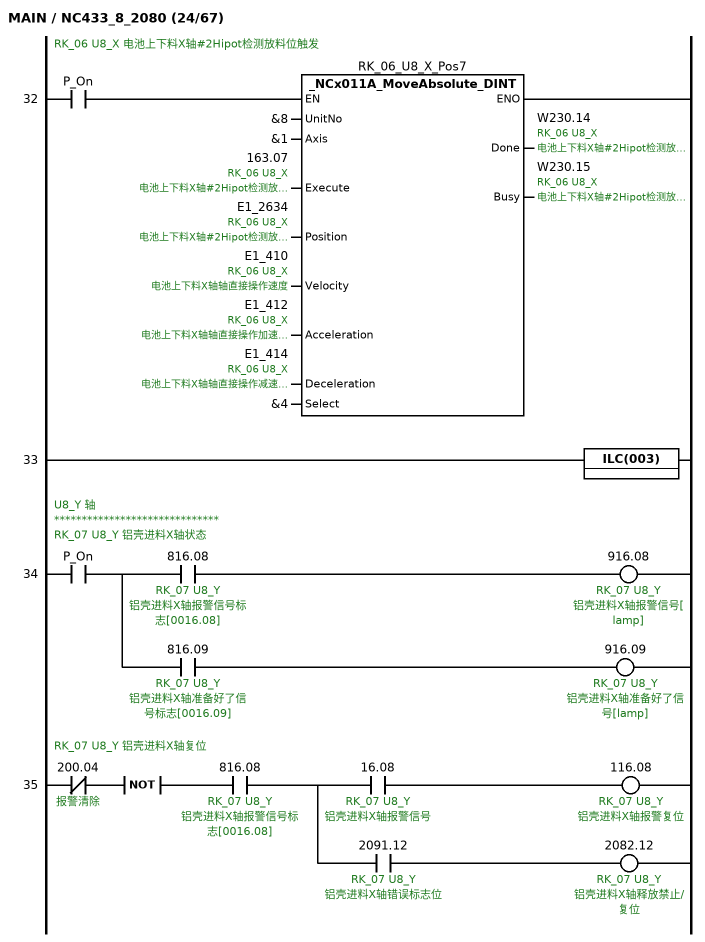
; [picture p288: MAIN / NC433_8_2080, rungs 32-35]
; rung 32: RK_06 U8_X 电池上下料X轴#2Hipot检测放料位触发
LD P_On
CALL RK_06_U8_X_Pos7 : _NCx011A_MoveAbsolute_DINT (UnitNo := &8, Axis := &1, Execute := 163.07, Position := E1_2634, Velocity := E1_410, Acceleration := E1_412, Deceleration := E1_414, Select := &4, Done => W230.14, Busy => W230.15)  ; RK_06 U8_X 电池上下料X轴#2Hipot检测放料位触发, RK_06 U8_X 电池上下料X轴#2Hipot检测放料位, RK_06 U8_X 电池上下料X轴轴直接操作速度, RK_06 U8_X 电池上下料X轴轴直接操作加速时间, RK_06 U8_X 电池上下料X轴轴直接操作减速时间, RK_06 U8_X 电池上下料X轴#2Hipot检测放料位完成标志, RK_06 U8_X 电池上下料X轴#2Hipot检测放料位忙标志
; rung 33
ILC(003)
; rung 34: U8_Y 轴 / ****************************** / RK_07 U8_Y 铝壳进料X轴状态
LD P_On
OUT TR0
AND 816.08  ; RK_07 U8_Y 铝壳进料X轴报警信号标志[0016.08]
OUT 916.08  ; RK_07 U8_Y 铝壳进料X轴报警信号[lamp]
LD TR0
AND 816.09  ; RK_07 U8_Y 铝壳进料X轴准备好了信号标志[0016.09]
OUT 916.09  ; RK_07 U8_Y 铝壳进料X轴准备好了信号[lamp]
; rung 35: RK_07 U8_Y 铝壳进料X轴复位
LDNOT 200.04  ; 报警清除
NOT(520)
AND 816.08  ; RK_07 U8_Y 铝壳进料X轴报警信号标志[0016.08]
OUT TR0
AND 16.08  ; RK_07 U8_Y 铝壳进料X轴报警信号
OUT 116.08  ; RK_07 U8_Y 铝壳进料X轴报警复位
LD TR0
AND 2091.12  ; RK_07 U8_Y 铝壳进料X轴错误标志位
OUT 2082.12  ; RK_07 U8_Y 铝壳进料X轴释放禁止/复位

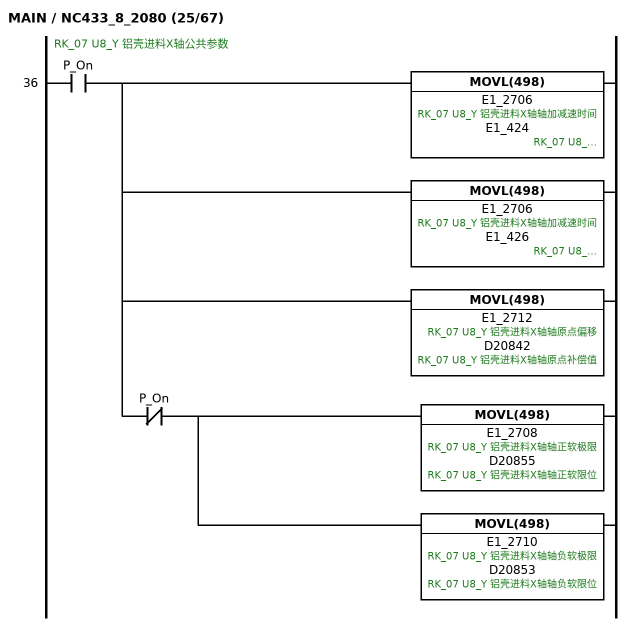
; rung 36: RK_07 U8_Y 铝壳进料X轴公共参数
LD P_On
MOVL(498) E1_2706 E1_424  ; RK_07 U8_Y 铝壳进料X轴轴加减速时间, RK_07 U8_Y 铝壳进料X轴轴直接操作加速时间
MOVL(498) E1_2706 E1_426  ; RK_07 U8_Y 铝壳进料X轴轴加减速时间, RK_07 U8_Y 铝壳进料X轴轴直接操作减速时间
MOVL(498) E1_2712 D20842  ; RK_07 U8_Y 铝壳进料X轴轴原点偏移, RK_07 U8_Y 铝壳进料X轴轴原点补偿值
ANDNOT P_On
MOVL(498) E1_2708 D20855  ; RK_07 U8_Y 铝壳进料X轴轴正软极限, RK_07 U8_Y 铝壳进料X轴轴正软限位
MOVL(498) E1_2710 D20853  ; RK_07 U8_Y 铝壳进料X轴轴负软极限, RK_07 U8_Y 铝壳进料X轴轴负软限位

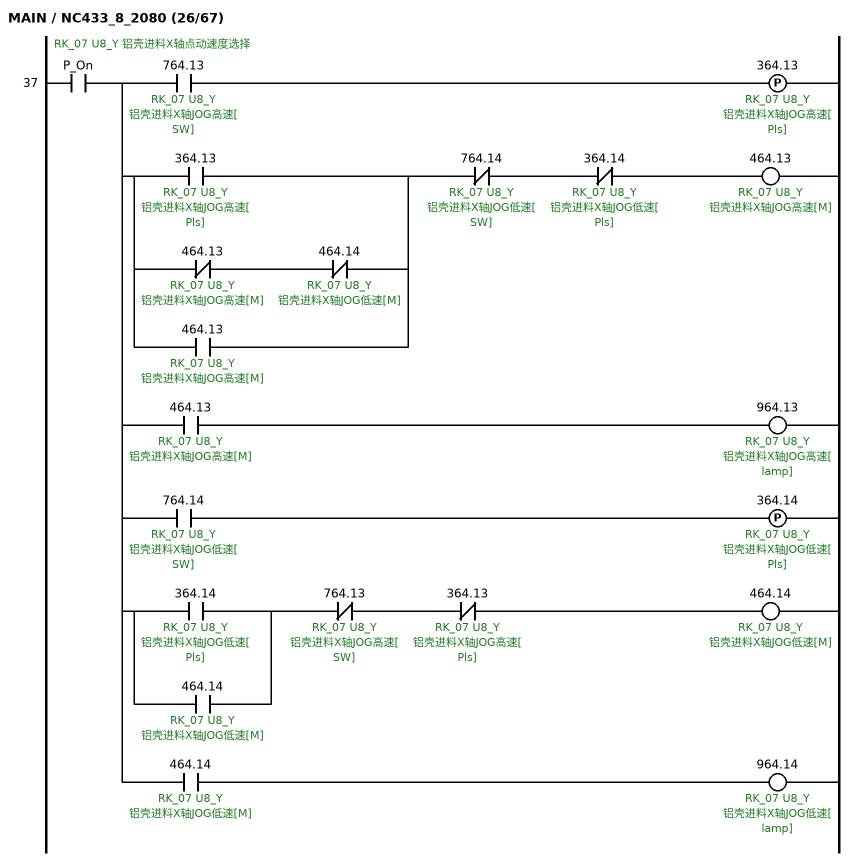
; rung 37: RK_07 U8_Y 铝壳进料X轴点动速度选择
LD P_On
OUT TR0
AND 764.13  ; RK_07 U8_Y 铝壳进料X轴JOG高速[SW]
DIFU(013) 364.13  ; RK_07 U8_Y 铝壳进料X轴JOG高速[Pls]
LD TR0
LD 364.13  ; RK_07 U8_Y 铝壳进料X轴JOG高速[Pls]
LDNOT 464.13  ; RK_07 U8_Y 铝壳进料X轴JOG高速[M]
ANDNOT 464.14  ; RK_07 U8_Y 铝壳进料X轴JOG低速[M]
ORLD
OR 464.13  ; RK_07 U8_Y 铝壳进料X轴JOG高速[M]
ANDLD
ANDNOT 764.14  ; RK_07 U8_Y 铝壳进料X轴JOG低速[SW]
ANDNOT 364.14  ; RK_07 U8_Y 铝壳进料X轴JOG低速[Pls]
OUT 464.13  ; RK_07 U8_Y 铝壳进料X轴JOG高速[M]
LD TR0
AND 464.13  ; RK_07 U8_Y 铝壳进料X轴JOG高速[M]
OUT 964.13  ; RK_07 U8_Y 铝壳进料X轴JOG高速[lamp]
LD TR0
AND 764.14  ; RK_07 U8_Y 铝壳进料X轴JOG低速[SW]
DIFU(013) 364.14  ; RK_07 U8_Y 铝壳进料X轴JOG低速[Pls]
LD TR0
LD 364.14  ; RK_07 U8_Y 铝壳进料X轴JOG低速[Pls]
OR 464.14  ; RK_07 U8_Y 铝壳进料X轴JOG低速[M]
ANDLD
ANDNOT 764.13  ; RK_07 U8_Y 铝壳进料X轴JOG高速[SW]
ANDNOT 364.13  ; RK_07 U8_Y 铝壳进料X轴JOG高速[Pls]
OUT 464.14  ; RK_07 U8_Y 铝壳进料X轴JOG低速[M]
LD TR0
AND 464.14  ; RK_07 U8_Y 铝壳进料X轴JOG低速[M]
OUT 964.14  ; RK_07 U8_Y 铝壳进料X轴JOG低速[lamp]

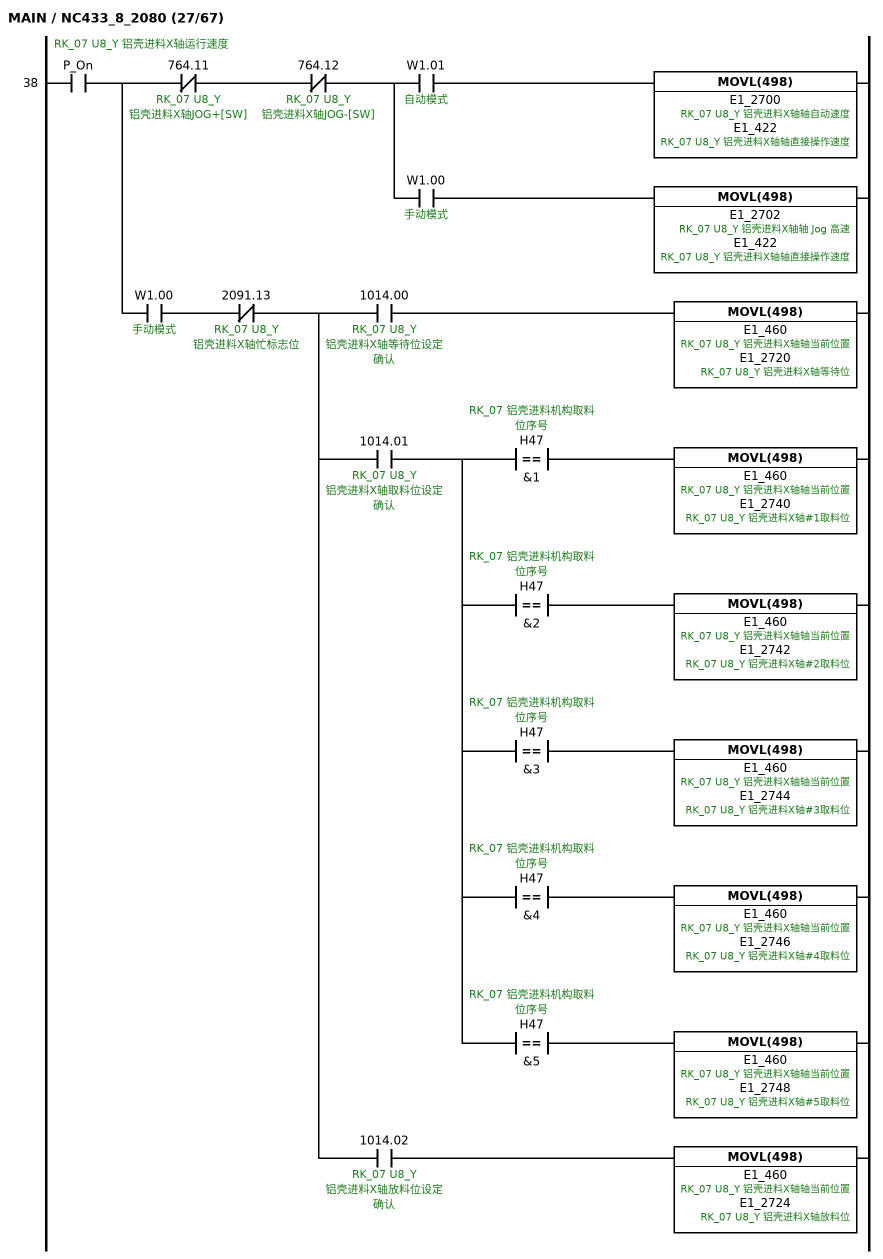
; rung 38: RK_07 U8_Y 铝壳进料X轴运行速度
LD P_On
OUT TR0
ANDNOT 764.11  ; RK_07 U8_Y 铝壳进料X轴JOG+[SW]
ANDNOT 764.12  ; RK_07 U8_Y 铝壳进料X轴JOG-[SW]
OUT TR1
AND W1.01  ; 自动模式
MOVL(498) E1_2700 E1_422  ; RK_07 U8_Y 铝壳进料X轴轴自动速度, RK_07 U8_Y 铝壳进料X轴轴直接操作速度
LD TR1
AND W1.00  ; 手动模式
MOVL(498) E1_2702 E1_422  ; RK_07 U8_Y 铝壳进料X轴轴 Jog 高速, RK_07 U8_Y 铝壳进料X轴轴直接操作速度
LD TR0
AND W1.00  ; 手动模式
ANDNOT 2091.13  ; RK_07 U8_Y 铝壳进料X轴忙标志位
OUT TR0
AND 1014.00  ; RK_07 U8_Y 铝壳进料X轴等待位设定确认
MOVL(498) E1_460 E1_2720  ; RK_07 U8_Y 铝壳进料X轴轴当前位置, RK_07 U8_Y 铝壳进料X轴等待位
LD TR0
AND 1014.01  ; RK_07 U8_Y 铝壳进料X轴取料位设定确认
OUT TR1
AND=(300) H47 &1  ; RK_07 铝壳进料机构取料位序号
MOVL(498) E1_460 E1_2740  ; RK_07 U8_Y 铝壳进料X轴轴当前位置, RK_07 U8_Y 铝壳进料X轴#1取料位
LD TR1
AND=(300) H47 &2  ; RK_07 铝壳进料机构取料位序号
MOVL(498) E1_460 E1_2742  ; RK_07 U8_Y 铝壳进料X轴轴当前位置, RK_07 U8_Y 铝壳进料X轴#2取料位
LD TR1
AND=(300) H47 &3  ; RK_07 铝壳进料机构取料位序号
MOVL(498) E1_460 E1_2744  ; RK_07 U8_Y 铝壳进料X轴轴当前位置, RK_07 U8_Y 铝壳进料X轴#3取料位
LD TR1
AND=(300) H47 &4  ; RK_07 铝壳进料机构取料位序号
MOVL(498) E1_460 E1_2746  ; RK_07 U8_Y 铝壳进料X轴轴当前位置, RK_07 U8_Y 铝壳进料X轴#4取料位
LD TR1
AND=(300) H47 &5  ; RK_07 铝壳进料机构取料位序号
MOVL(498) E1_460 E1_2748  ; RK_07 U8_Y 铝壳进料X轴轴当前位置, RK_07 U8_Y 铝壳进料X轴#5取料位
LD TR0
AND 1014.02  ; RK_07 U8_Y 铝壳进料X轴放料位设定确认
MOVL(498) E1_460 E1_2724  ; RK_07 U8_Y 铝壳进料X轴轴当前位置, RK_07 U8_Y 铝壳进料X轴放料位

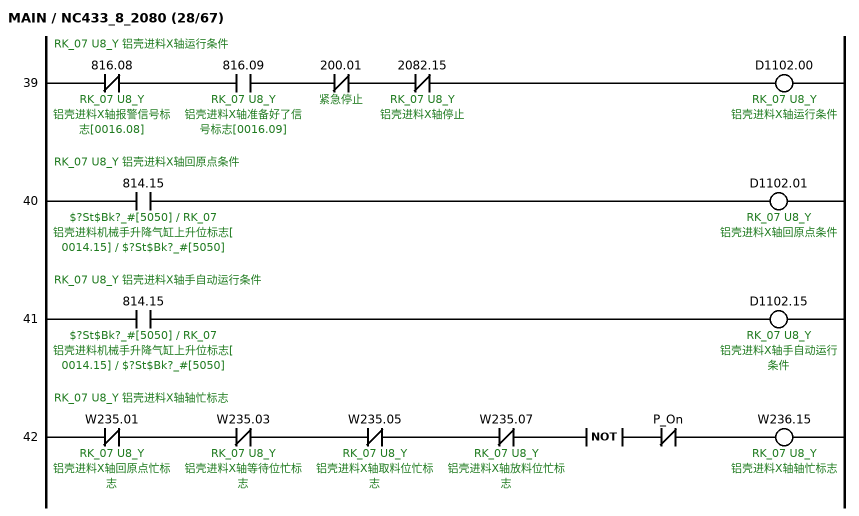
; rung 39: RK_07 U8_Y 铝壳进料X轴运行条件
LDNOT 816.08  ; RK_07 U8_Y 铝壳进料X轴报警信号标志[0016.08]
AND 816.09  ; RK_07 U8_Y 铝壳进料X轴准备好了信号标志[0016.09]
ANDNOT 200.01  ; 紧急停止
ANDNOT 2082.15  ; RK_07 U8_Y 铝壳进料X轴停止
OUT D1102.00  ; RK_07 U8_Y 铝壳进料X轴运行条件
; rung 40: RK_07 U8_Y 铝壳进料X轴回原点条件
LD 814.15  ; $?St$Bk?_#[5050] / RK_07 铝壳进料机械手升降气缸上升位标志[0014.15] / $?St$Bk?_#[5050]
OUT D1102.01  ; RK_07 U8_Y 铝壳进料X轴回原点条件
; rung 41: RK_07 U8_Y 铝壳进料X轴手自动运行条件
LD 814.15  ; $?St$Bk?_#[5050] / RK_07 铝壳进料机械手升降气缸上升位标志[0014.15] / $?St$Bk?_#[5050]
OUT D1102.15  ; RK_07 U8_Y 铝壳进料X轴手自动运行条件
; rung 42: RK_07 U8_Y 铝壳进料X轴轴忙标志
LDNOT W235.01  ; RK_07 U8_Y 铝壳进料X轴回原点忙标志
ANDNOT W235.03  ; RK_07 U8_Y 铝壳进料X轴等待位忙标志
ANDNOT W235.05  ; RK_07 U8_Y 铝壳进料X轴取料位忙标志
ANDNOT W235.07  ; RK_07 U8_Y 铝壳进料X轴放料位忙标志
NOT(520)
ANDNOT P_On
OUT W236.15  ; RK_07 U8_Y 铝壳进料X轴轴忙标志

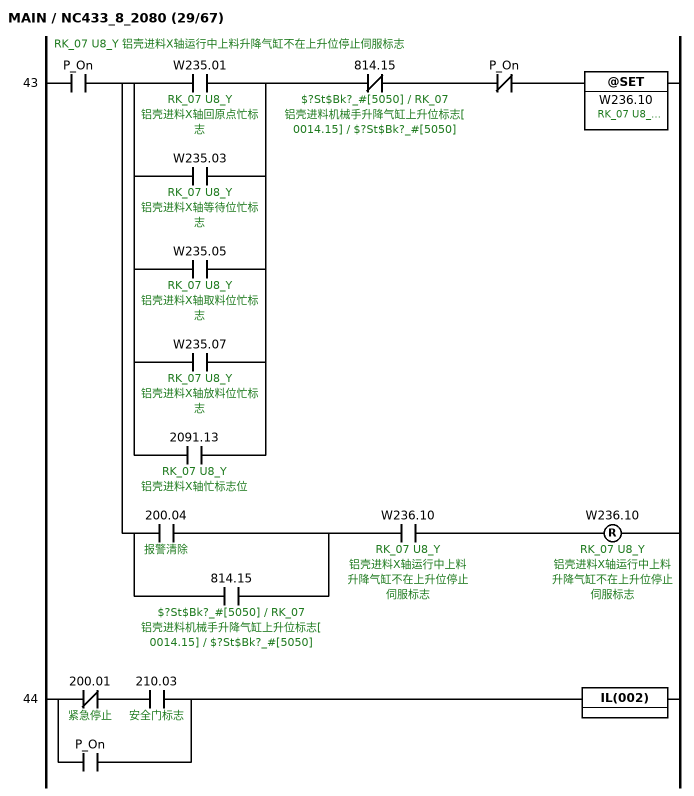
; rung 43: RK_07 U8_Y 铝壳进料X轴运行中上料升降气缸不在上升位停止伺服标志
LD P_On
OUT TR0
LD W235.01  ; RK_07 U8_Y 铝壳进料X轴回原点忙标志
OR W235.03  ; RK_07 U8_Y 铝壳进料X轴等待位忙标志
OR W235.05  ; RK_07 U8_Y 铝壳进料X轴取料位忙标志
OR W235.07  ; RK_07 U8_Y 铝壳进料X轴放料位忙标志
OR 2091.13  ; RK_07 U8_Y 铝壳进料X轴忙标志位
ANDLD
ANDNOT 814.15  ; $?St$Bk?_#[5050] / RK_07 铝壳进料机械手升降气缸上升位标志[0014.15] / $?St$Bk?_#[5050]
ANDNOT P_On
@SET W236.10  ; RK_07 U8_Y 铝壳进料X轴运行中上料升降气缸不在上升位停止伺服标志  // 增加相应报警信息
LD TR0
LD 200.04  ; 报警清除
OR 814.15  ; $?St$Bk?_#[5050] / RK_07 铝壳进料机械手升降气缸上升位标志[0014.15] / $?St$Bk?_#[5050]
ANDLD
AND W236.10  ; RK_07 U8_Y 铝壳进料X轴运行中上料升降气缸不在上升位停止伺服标志
RSET W236.10  ; RK_07 U8_Y 铝壳进料X轴运行中上料升降气缸不在上升位停止伺服标志
; rung 44
LDNOT 200.01  ; 紧急停止
AND 210.03  ; 安全门标志
OR P_On
IL(002)

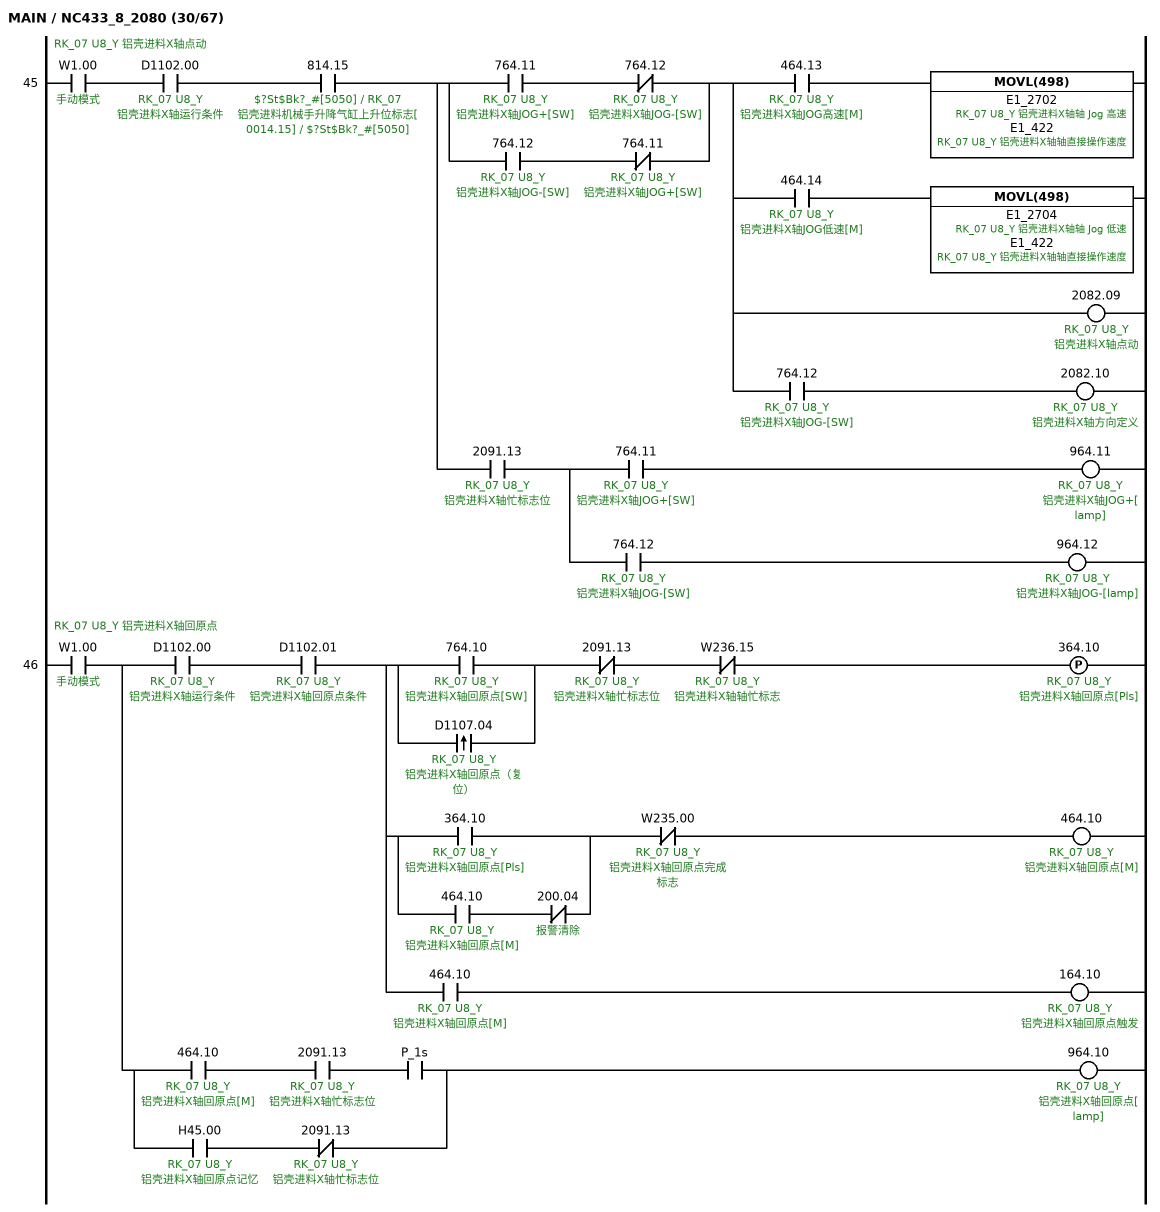
; rung 45: RK_07 U8_Y 铝壳进料X轴点动
LD W1.00  ; 手动模式
AND D1102.00  ; RK_07 U8_Y 铝壳进料X轴运行条件
AND 814.15  ; $?St$Bk?_#[5050] / RK_07 铝壳进料机械手升降气缸上升位标志[0014.15] / $?St$Bk?_#[5050]
OUT TR0
LD 764.11  ; RK_07 U8_Y 铝壳进料X轴JOG+[SW]
ANDNOT 764.12  ; RK_07 U8_Y 铝壳进料X轴JOG-[SW]
LD 764.12  ; RK_07 U8_Y 铝壳进料X轴JOG-[SW]
ANDNOT 764.11  ; RK_07 U8_Y 铝壳进料X轴JOG+[SW]
ORLD
ANDLD
OUT TR1
AND 464.13  ; RK_07 U8_Y 铝壳进料X轴JOG高速[M]
MOVL(498) E1_2702 E1_422  ; RK_07 U8_Y 铝壳进料X轴轴 Jog 高速, RK_07 U8_Y 铝壳进料X轴轴直接操作速度
LD TR1
AND 464.14  ; RK_07 U8_Y 铝壳进料X轴JOG低速[M]
MOVL(498) E1_2704 E1_422  ; RK_07 U8_Y 铝壳进料X轴轴 Jog 低速, RK_07 U8_Y 铝壳进料X轴轴直接操作速度
LD TR1
OUT 2082.09  ; RK_07 U8_Y 铝壳进料X轴点动
AND 764.12  ; RK_07 U8_Y 铝壳进料X轴JOG-[SW]
OUT 2082.10  ; RK_07 U8_Y 铝壳进料X轴方向定义
LD TR0
AND 2091.13  ; RK_07 U8_Y 铝壳进料X轴忙标志位
OUT TR0
AND 764.11  ; RK_07 U8_Y 铝壳进料X轴JOG+[SW]
OUT 964.11  ; RK_07 U8_Y 铝壳进料X轴JOG+[lamp]
LD TR0
AND 764.12  ; RK_07 U8_Y 铝壳进料X轴JOG-[SW]
OUT 964.12  ; RK_07 U8_Y 铝壳进料X轴JOG-[lamp]
; rung 46: RK_07 U8_Y 铝壳进料X轴回原点
LD W1.00  ; 手动模式
OUT TR0
AND D1102.00  ; RK_07 U8_Y 铝壳进料X轴运行条件
AND D1102.01  ; RK_07 U8_Y 铝壳进料X轴回原点条件
OUT TR1
LD 764.10  ; RK_07 U8_Y 铝壳进料X轴回原点[SW]
@OR D1107.04  ; RK_07 U8_Y 铝壳进料X轴回原点（复位）
ANDLD
ANDNOT 2091.13  ; RK_07 U8_Y 铝壳进料X轴忙标志位
ANDNOT W236.15  ; RK_07 U8_Y 铝壳进料X轴轴忙标志
DIFU(013) 364.10  ; RK_07 U8_Y 铝壳进料X轴回原点[Pls]
LD TR1
LD 364.10  ; RK_07 U8_Y 铝壳进料X轴回原点[Pls]
LD 464.10  ; RK_07 U8_Y 铝壳进料X轴回原点[M]
ANDNOT 200.04  ; 报警清除
ORLD
ANDLD
ANDNOT W235.00  ; RK_07 U8_Y 铝壳进料X轴回原点完成标志
OUT 464.10  ; RK_07 U8_Y 铝壳进料X轴回原点[M]
LD TR1
AND 464.10  ; RK_07 U8_Y 铝壳进料X轴回原点[M]
OUT 164.10  ; RK_07 U8_Y 铝壳进料X轴回原点触发
LD TR0
LD 464.10  ; RK_07 U8_Y 铝壳进料X轴回原点[M]
AND 2091.13  ; RK_07 U8_Y 铝壳进料X轴忙标志位
AND P_1s
LD H45.00  ; RK_07 U8_Y 铝壳进料X轴回原点记忆
ANDNOT 2091.13  ; RK_07 U8_Y 铝壳进料X轴忙标志位
ORLD
ANDLD
OUT 964.10  ; RK_07 U8_Y 铝壳进料X轴回原点[lamp]

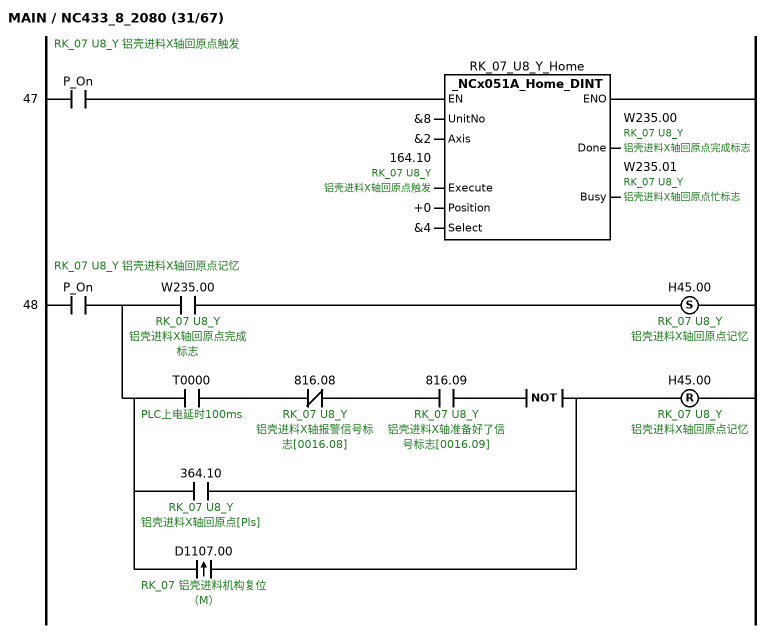
; rung 47: RK_07 U8_Y 铝壳进料X轴回原点触发
LD P_On
CALL RK_07_U8_Y_Home : _NCx051A_Home_DINT (UnitNo := &8, Axis := &2, Execute := 164.10, Position := +0, Select := &4, Done => W235.00, Busy => W235.01)  ; RK_07 U8_Y 铝壳进料X轴回原点触发, RK_07 U8_Y 铝壳进料X轴回原点完成标志, RK_07 U8_Y 铝壳进料X轴回原点忙标志
; rung 48: RK_07 U8_Y 铝壳进料X轴回原点记忆
LD P_On
OUT TR0
AND W235.00  ; RK_07 U8_Y 铝壳进料X轴回原点完成标志
SET H45.00  ; RK_07 U8_Y 铝壳进料X轴回原点记忆
LD TR0
LD T0000  ; PLC上电延时100ms
ANDNOT 816.08  ; RK_07 U8_Y 铝壳进料X轴报警信号标志[0016.08]
AND 816.09  ; RK_07 U8_Y 铝壳进料X轴准备好了信号标志[0016.09]
NOT(520)
OR 364.10  ; RK_07 U8_Y 铝壳进料X轴回原点[Pls]
@OR D1107.00  ; RK_07 铝壳进料机构复位（M）
ANDLD
RSET H45.00  ; RK_07 U8_Y 铝壳进料X轴回原点记忆

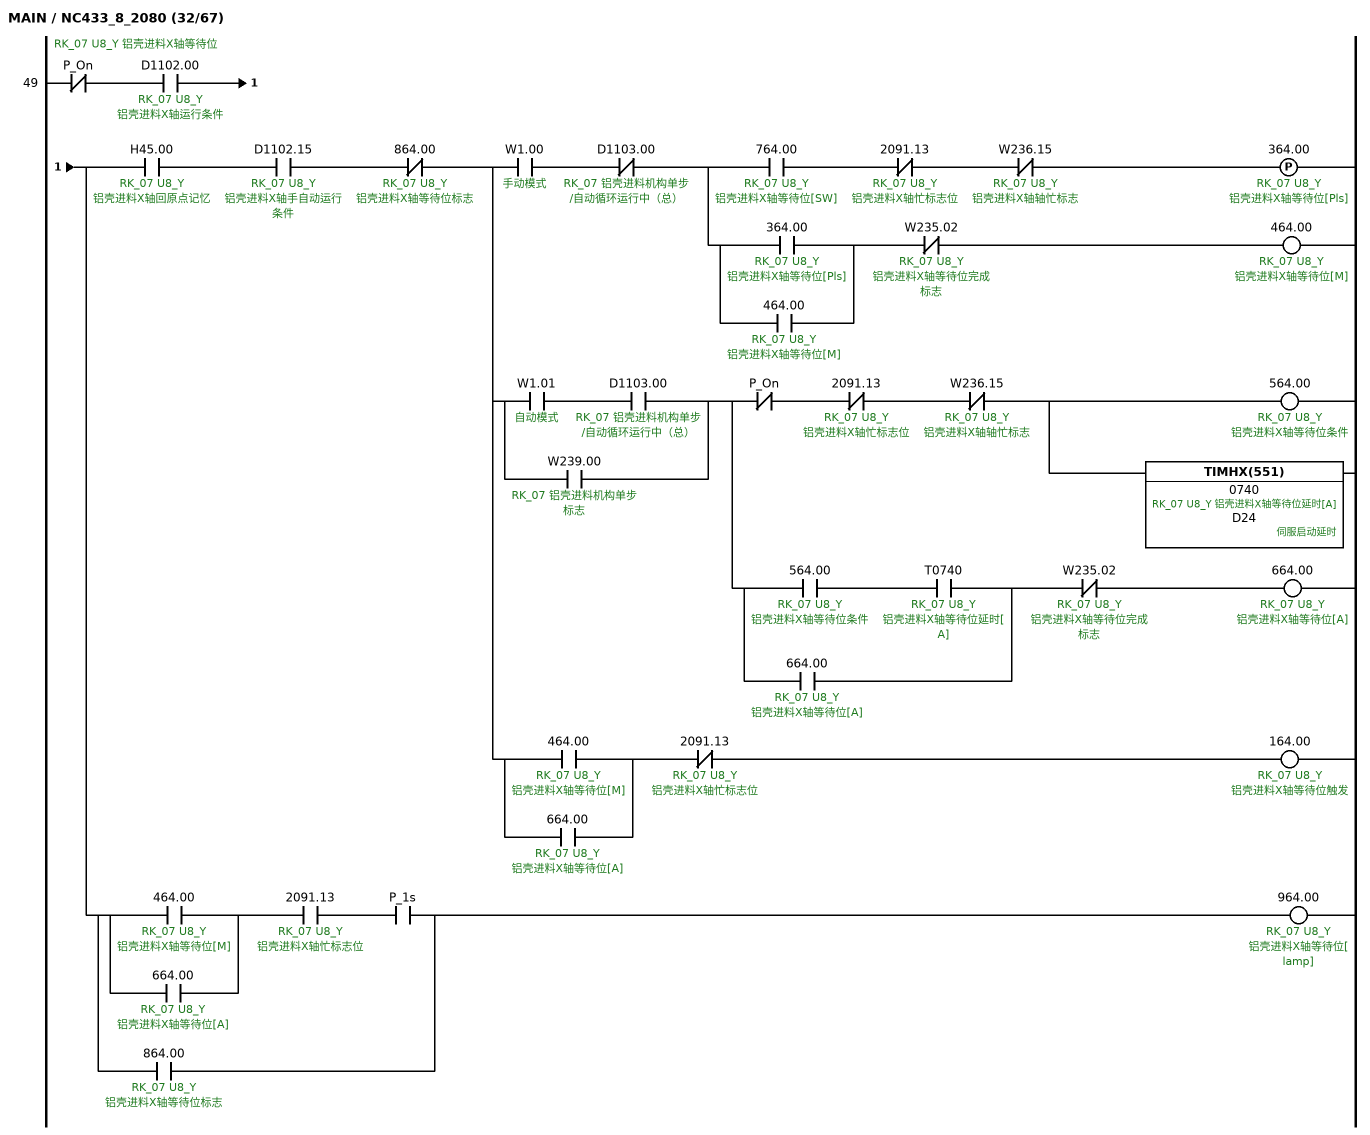
; rung 49: RK_07 U8_Y 铝壳进料X轴等待位
LDNOT P_On
AND D1102.00  ; RK_07 U8_Y 铝壳进料X轴运行条件
OUT TR0
AND H45.00  ; RK_07 U8_Y 铝壳进料X轴回原点记忆
AND D1102.15  ; RK_07 U8_Y 铝壳进料X轴手自动运行条件
ANDNOT 864.00  ; RK_07 U8_Y 铝壳进料X轴等待位标志
OUT TR1
AND W1.00  ; 手动模式
ANDNOT D1103.00  ; RK_07 铝壳进料机构单步/自动循环运行中（总）
OUT TR2
AND 764.00  ; RK_07 U8_Y 铝壳进料X轴等待位[SW]
ANDNOT 2091.13  ; RK_07 U8_Y 铝壳进料X轴忙标志位
ANDNOT W236.15  ; RK_07 U8_Y 铝壳进料X轴轴忙标志
DIFU(013) 364.00  ; RK_07 U8_Y 铝壳进料X轴等待位[Pls]
LD TR2
LD 364.00  ; RK_07 U8_Y 铝壳进料X轴等待位[Pls]
OR 464.00  ; RK_07 U8_Y 铝壳进料X轴等待位[M]
ANDLD
ANDNOT W235.02  ; RK_07 U8_Y 铝壳进料X轴等待位完成标志
OUT 464.00  ; RK_07 U8_Y 铝壳进料X轴等待位[M]
LD TR1
LD W1.01  ; 自动模式
AND D1103.00  ; RK_07 铝壳进料机构单步/自动循环运行中（总）
OR W239.00  ; RK_07 铝壳进料机构单步标志
ANDLD
OUT TR2
ANDNOT P_On  // RK_07 U8_Y 铝壳进料X轴等待位（步）
ANDNOT 2091.13  ; RK_07 U8_Y 铝壳进料X轴忙标志位
ANDNOT W236.15  ; RK_07 U8_Y 铝壳进料X轴轴忙标志
OUT 564.00  ; RK_07 U8_Y 铝壳进料X轴等待位条件
TIMHX(551) 0740 D24  ; 伺服启动延时, RK_07 U8_Y 铝壳进料X轴等待位延时[A]
LD TR2
LD 564.00  ; RK_07 U8_Y 铝壳进料X轴等待位条件
AND T0740  ; RK_07 U8_Y 铝壳进料X轴等待位延时[A]
OR 664.00  ; RK_07 U8_Y 铝壳进料X轴等待位[A]
ANDLD
ANDNOT W235.02  ; RK_07 U8_Y 铝壳进料X轴等待位完成标志
OUT 664.00  ; RK_07 U8_Y 铝壳进料X轴等待位[A]
LD TR1
LD 464.00  ; RK_07 U8_Y 铝壳进料X轴等待位[M]
OR 664.00  ; RK_07 U8_Y 铝壳进料X轴等待位[A]
ANDLD
ANDNOT 2091.13  ; RK_07 U8_Y 铝壳进料X轴忙标志位
OUT 164.00  ; RK_07 U8_Y 铝壳进料X轴等待位触发
LD TR0
LD 464.00  ; RK_07 U8_Y 铝壳进料X轴等待位[M]
OR 664.00  ; RK_07 U8_Y 铝壳进料X轴等待位[A]
AND 2091.13  ; RK_07 U8_Y 铝壳进料X轴忙标志位
AND P_1s
OR 864.00  ; RK_07 U8_Y 铝壳进料X轴等待位标志
ANDLD
OUT 964.00  ; RK_07 U8_Y 铝壳进料X轴等待位[lamp]

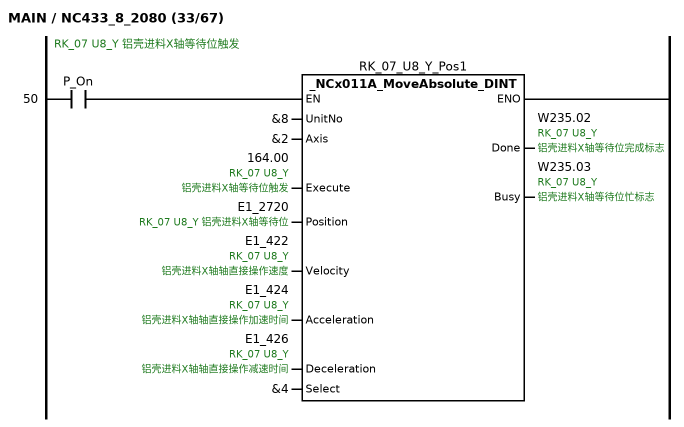
; rung 50: RK_07 U8_Y 铝壳进料X轴等待位触发
LD P_On
CALL RK_07_U8_Y_Pos1 : _NCx011A_MoveAbsolute_DINT (UnitNo := &8, Axis := &2, Execute := 164.00, Position := E1_2720, Velocity := E1_422, Acceleration := E1_424, Deceleration := E1_426, Select := &4, Done => W235.02, Busy => W235.03)  ; RK_07 U8_Y 铝壳进料X轴等待位触发, RK_07 U8_Y 铝壳进料X轴等待位, RK_07 U8_Y 铝壳进料X轴轴直接操作速度, RK_07 U8_Y 铝壳进料X轴轴直接操作加速时间, RK_07 U8_Y 铝壳进料X轴轴直接操作减速时间, RK_07 U8_Y 铝壳进料X轴等待位完成标志, RK_07 U8_Y 铝壳进料X轴等待位忙标志

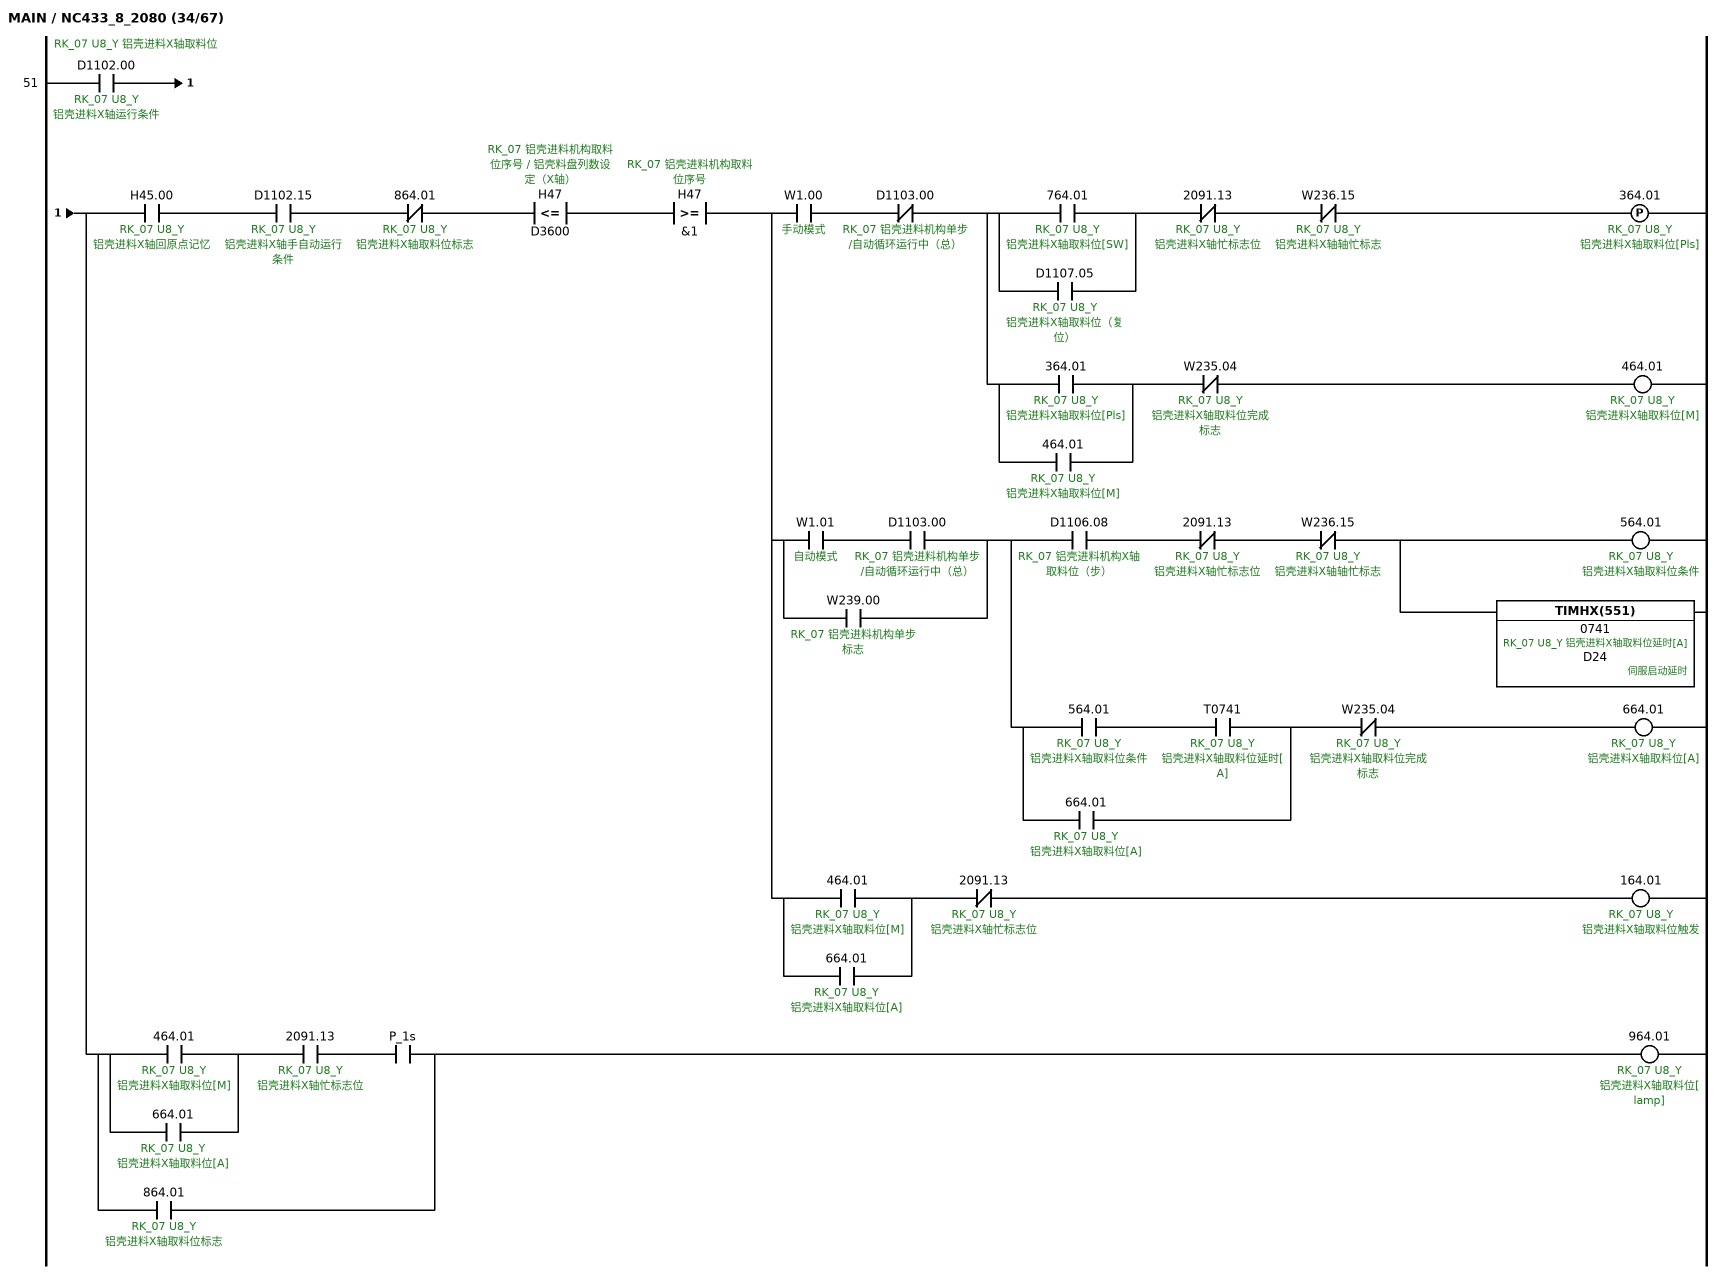
; rung 51: RK_07 U8_Y 铝壳进料X轴取料位
LD D1102.00  ; RK_07 U8_Y 铝壳进料X轴运行条件
OUT TR0
AND H45.00  ; RK_07 U8_Y 铝壳进料X轴回原点记忆
AND D1102.15  ; RK_07 U8_Y 铝壳进料X轴手自动运行条件
ANDNOT 864.01  ; RK_07 U8_Y 铝壳进料X轴取料位标志
AND<=(315) H47 D3600  ; RK_07 铝壳进料机构取料位序号, 铝壳料盘列数设定（X轴）
AND>=(325) H47 &1  ; RK_07 铝壳进料机构取料位序号
OUT TR1
AND W1.00  ; 手动模式
ANDNOT D1103.00  ; RK_07 铝壳进料机构单步/自动循环运行中（总）
OUT TR2
LD 764.01  ; RK_07 U8_Y 铝壳进料X轴取料位[SW]
OR D1107.05  ; RK_07 U8_Y 铝壳进料X轴取料位（复位）
ANDLD
ANDNOT 2091.13  ; RK_07 U8_Y 铝壳进料X轴忙标志位
ANDNOT W236.15  ; RK_07 U8_Y 铝壳进料X轴轴忙标志
DIFU(013) 364.01  ; RK_07 U8_Y 铝壳进料X轴取料位[Pls]
LD TR2
LD 364.01  ; RK_07 U8_Y 铝壳进料X轴取料位[Pls]
OR 464.01  ; RK_07 U8_Y 铝壳进料X轴取料位[M]
ANDLD
ANDNOT W235.04  ; RK_07 U8_Y 铝壳进料X轴取料位完成标志
OUT 464.01  ; RK_07 U8_Y 铝壳进料X轴取料位[M]
LD TR1
LD W1.01  ; 自动模式
AND D1103.00  ; RK_07 铝壳进料机构单步/自动循环运行中（总）
OR W239.00  ; RK_07 铝壳进料机构单步标志
ANDLD
OUT TR2
AND D1106.08  ; RK_07 铝壳进料机构X轴取料位（步）
ANDNOT 2091.13  ; RK_07 U8_Y 铝壳进料X轴忙标志位
ANDNOT W236.15  ; RK_07 U8_Y 铝壳进料X轴轴忙标志
OUT 564.01  ; RK_07 U8_Y 铝壳进料X轴取料位条件
TIMHX(551) 0741 D24  ; 伺服启动延时, RK_07 U8_Y 铝壳进料X轴取料位延时[A]
LD TR2
LD 564.01  ; RK_07 U8_Y 铝壳进料X轴取料位条件
AND T0741  ; RK_07 U8_Y 铝壳进料X轴取料位延时[A]
OR 664.01  ; RK_07 U8_Y 铝壳进料X轴取料位[A]
ANDLD
ANDNOT W235.04  ; RK_07 U8_Y 铝壳进料X轴取料位完成标志
OUT 664.01  ; RK_07 U8_Y 铝壳进料X轴取料位[A]
LD TR1
LD 464.01  ; RK_07 U8_Y 铝壳进料X轴取料位[M]
OR 664.01  ; RK_07 U8_Y 铝壳进料X轴取料位[A]
ANDLD
ANDNOT 2091.13  ; RK_07 U8_Y 铝壳进料X轴忙标志位
OUT 164.01  ; RK_07 U8_Y 铝壳进料X轴取料位触发
LD TR0
LD 464.01  ; RK_07 U8_Y 铝壳进料X轴取料位[M]
OR 664.01  ; RK_07 U8_Y 铝壳进料X轴取料位[A]
AND 2091.13  ; RK_07 U8_Y 铝壳进料X轴忙标志位
AND P_1s
OR 864.01  ; RK_07 U8_Y 铝壳进料X轴取料位标志
ANDLD
OUT 964.01  ; RK_07 U8_Y 铝壳进料X轴取料位[lamp]

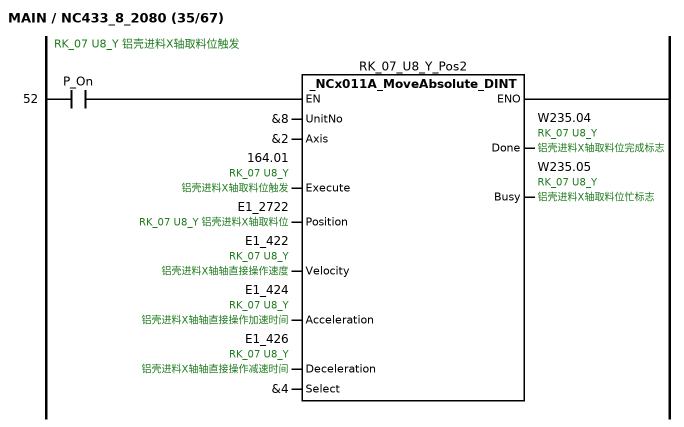
; rung 52: RK_07 U8_Y 铝壳进料X轴取料位触发
LD P_On
CALL RK_07_U8_Y_Pos2 : _NCx011A_MoveAbsolute_DINT (UnitNo := &8, Axis := &2, Execute := 164.01, Position := E1_2722, Velocity := E1_422, Acceleration := E1_424, Deceleration := E1_426, Select := &4, Done => W235.04, Busy => W235.05)  ; RK_07 U8_Y 铝壳进料X轴取料位触发, RK_07 U8_Y 铝壳进料X轴取料位, RK_07 U8_Y 铝壳进料X轴轴直接操作速度, RK_07 U8_Y 铝壳进料X轴轴直接操作加速时间, RK_07 U8_Y 铝壳进料X轴轴直接操作减速时间, RK_07 U8_Y 铝壳进料X轴取料位完成标志, RK_07 U8_Y 铝壳进料X轴取料位忙标志

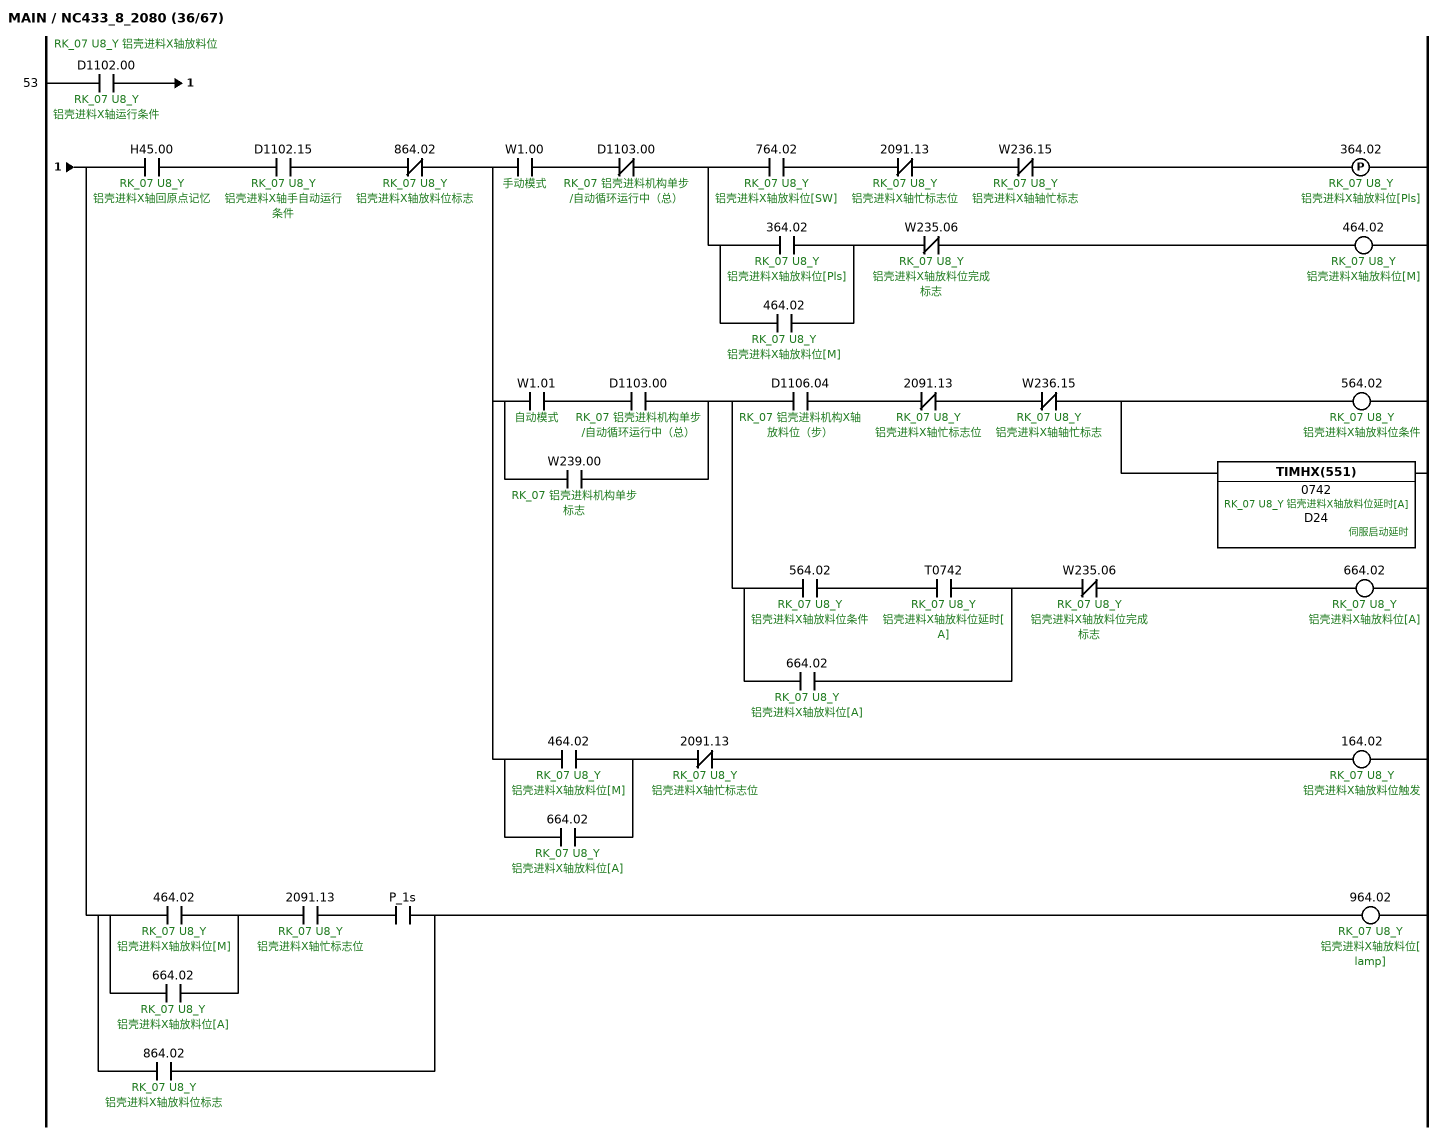
; rung 53: RK_07 U8_Y 铝壳进料X轴放料位
LD D1102.00  ; RK_07 U8_Y 铝壳进料X轴运行条件
OUT TR0
AND H45.00  ; RK_07 U8_Y 铝壳进料X轴回原点记忆
AND D1102.15  ; RK_07 U8_Y 铝壳进料X轴手自动运行条件
ANDNOT 864.02  ; RK_07 U8_Y 铝壳进料X轴放料位标志
OUT TR1
AND W1.00  ; 手动模式
ANDNOT D1103.00  ; RK_07 铝壳进料机构单步/自动循环运行中（总）
OUT TR2
AND 764.02  ; RK_07 U8_Y 铝壳进料X轴放料位[SW]
ANDNOT 2091.13  ; RK_07 U8_Y 铝壳进料X轴忙标志位
ANDNOT W236.15  ; RK_07 U8_Y 铝壳进料X轴轴忙标志
DIFU(013) 364.02  ; RK_07 U8_Y 铝壳进料X轴放料位[Pls]
LD TR2
LD 364.02  ; RK_07 U8_Y 铝壳进料X轴放料位[Pls]
OR 464.02  ; RK_07 U8_Y 铝壳进料X轴放料位[M]
ANDLD
ANDNOT W235.06  ; RK_07 U8_Y 铝壳进料X轴放料位完成标志
OUT 464.02  ; RK_07 U8_Y 铝壳进料X轴放料位[M]
LD TR1
LD W1.01  ; 自动模式
AND D1103.00  ; RK_07 铝壳进料机构单步/自动循环运行中（总）
OR W239.00  ; RK_07 铝壳进料机构单步标志
ANDLD
OUT TR2
AND D1106.04  ; RK_07 铝壳进料机构X轴放料位（步）
ANDNOT 2091.13  ; RK_07 U8_Y 铝壳进料X轴忙标志位
ANDNOT W236.15  ; RK_07 U8_Y 铝壳进料X轴轴忙标志
OUT 564.02  ; RK_07 U8_Y 铝壳进料X轴放料位条件
TIMHX(551) 0742 D24  ; 伺服启动延时, RK_07 U8_Y 铝壳进料X轴放料位延时[A]
LD TR2
LD 564.02  ; RK_07 U8_Y 铝壳进料X轴放料位条件
AND T0742  ; RK_07 U8_Y 铝壳进料X轴放料位延时[A]
OR 664.02  ; RK_07 U8_Y 铝壳进料X轴放料位[A]
ANDLD
ANDNOT W235.06  ; RK_07 U8_Y 铝壳进料X轴放料位完成标志
OUT 664.02  ; RK_07 U8_Y 铝壳进料X轴放料位[A]
LD TR1
LD 464.02  ; RK_07 U8_Y 铝壳进料X轴放料位[M]
OR 664.02  ; RK_07 U8_Y 铝壳进料X轴放料位[A]
ANDLD
ANDNOT 2091.13  ; RK_07 U8_Y 铝壳进料X轴忙标志位
OUT 164.02  ; RK_07 U8_Y 铝壳进料X轴放料位触发
LD TR0
LD 464.02  ; RK_07 U8_Y 铝壳进料X轴放料位[M]
OR 664.02  ; RK_07 U8_Y 铝壳进料X轴放料位[A]
AND 2091.13  ; RK_07 U8_Y 铝壳进料X轴忙标志位
AND P_1s
OR 864.02  ; RK_07 U8_Y 铝壳进料X轴放料位标志
ANDLD
OUT 964.02  ; RK_07 U8_Y 铝壳进料X轴放料位[lamp]

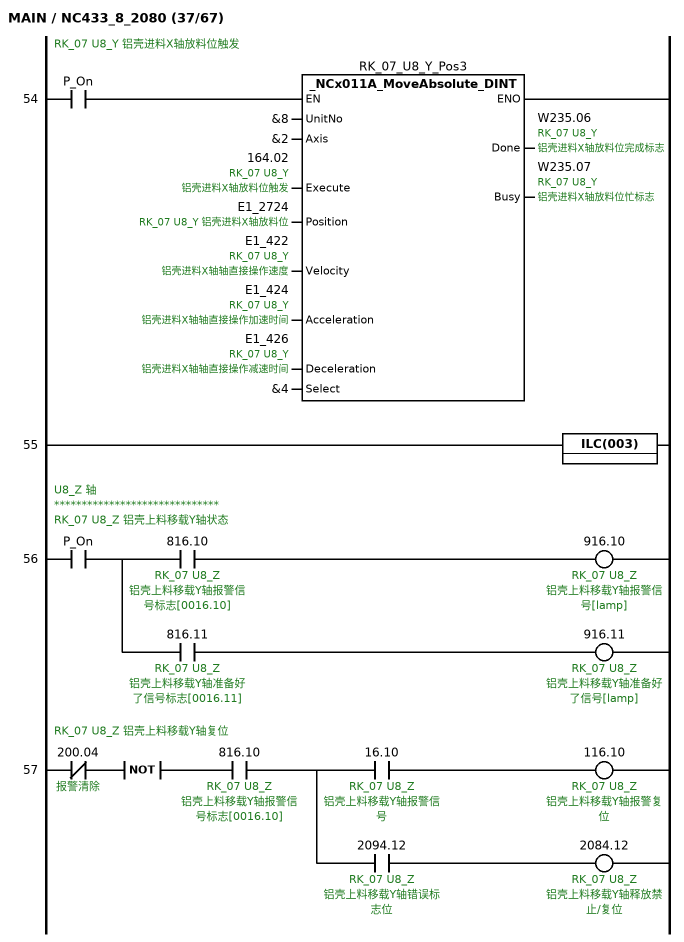
; rung 54: RK_07 U8_Y 铝壳进料X轴放料位触发
LD P_On
CALL RK_07_U8_Y_Pos3 : _NCx011A_MoveAbsolute_DINT (UnitNo := &8, Axis := &2, Execute := 164.02, Position := E1_2724, Velocity := E1_422, Acceleration := E1_424, Deceleration := E1_426, Select := &4, Done => W235.06, Busy => W235.07)  ; RK_07 U8_Y 铝壳进料X轴放料位触发, RK_07 U8_Y 铝壳进料X轴放料位, RK_07 U8_Y 铝壳进料X轴轴直接操作速度, RK_07 U8_Y 铝壳进料X轴轴直接操作加速时间, RK_07 U8_Y 铝壳进料X轴轴直接操作减速时间, RK_07 U8_Y 铝壳进料X轴放料位完成标志, RK_07 U8_Y 铝壳进料X轴放料位忙标志
; rung 55
ILC(003)
; rung 56: U8_Z 轴 / ****************************** / RK_07 U8_Z 铝壳上料移载Y轴状态
LD P_On
OUT TR0
AND 816.10  ; RK_07 U8_Z 铝壳上料移载Y轴报警信号标志[0016.10]
OUT 916.10  ; RK_07 U8_Z 铝壳上料移载Y轴报警信号[lamp]
LD TR0
AND 816.11  ; RK_07 U8_Z 铝壳上料移载Y轴准备好了信号标志[0016.11]
OUT 916.11  ; RK_07 U8_Z 铝壳上料移载Y轴准备好了信号[lamp]
; rung 57: RK_07 U8_Z 铝壳上料移载Y轴复位
LDNOT 200.04  ; 报警清除
NOT(520)
AND 816.10  ; RK_07 U8_Z 铝壳上料移载Y轴报警信号标志[0016.10]
OUT TR0
AND 16.10  ; RK_07 U8_Z 铝壳上料移载Y轴报警信号
OUT 116.10  ; RK_07 U8_Z 铝壳上料移载Y轴报警复位
LD TR0
AND 2094.12  ; RK_07 U8_Z 铝壳上料移载Y轴错误标志位
OUT 2084.12  ; RK_07 U8_Z 铝壳上料移载Y轴释放禁止/复位

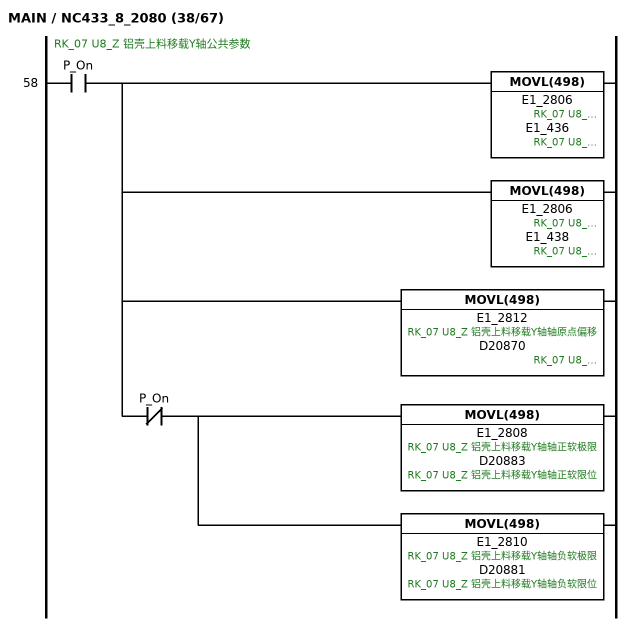
; rung 58: RK_07 U8_Z 铝壳上料移载Y轴公共参数
LD P_On
MOVL(498) E1_2806 E1_436  ; RK_07 U8_Z 铝壳上料移载Y轴轴加减速时间, RK_07 U8_Z 铝壳上料移载Y轴轴直接操作加速时间
MOVL(498) E1_2806 E1_438  ; RK_07 U8_Z 铝壳上料移载Y轴轴加减速时间, RK_07 U8_Z 铝壳上料移载Y轴轴直接操作减速时间
MOVL(498) E1_2812 D20870  ; RK_07 U8_Z 铝壳上料移载Y轴轴原点偏移, RK_07 U8_Z 铝壳上料移载Y轴轴原点补偿值
ANDNOT P_On
MOVL(498) E1_2808 D20883  ; RK_07 U8_Z 铝壳上料移载Y轴轴正软极限, RK_07 U8_Z 铝壳上料移载Y轴轴正软限位
MOVL(498) E1_2810 D20881  ; RK_07 U8_Z 铝壳上料移载Y轴轴负软极限, RK_07 U8_Z 铝壳上料移载Y轴轴负软限位

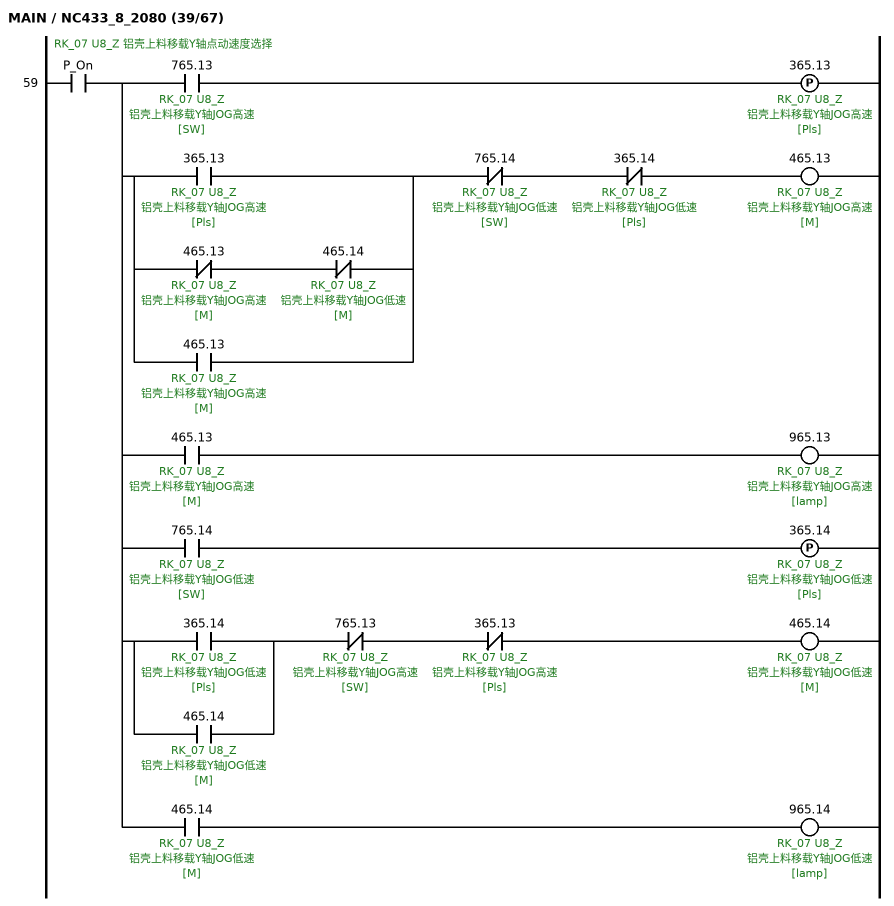
; rung 59: RK_07 U8_Z 铝壳上料移载Y轴点动速度选择
LD P_On
OUT TR0
AND 765.13  ; RK_07 U8_Z 铝壳上料移载Y轴JOG高速[SW]
DIFU(013) 365.13  ; RK_07 U8_Z 铝壳上料移载Y轴JOG高速[Pls]
LD TR0
LD 365.13  ; RK_07 U8_Z 铝壳上料移载Y轴JOG高速[Pls]
LDNOT 465.13  ; RK_07 U8_Z 铝壳上料移载Y轴JOG高速[M]
ANDNOT 465.14  ; RK_07 U8_Z 铝壳上料移载Y轴JOG低速[M]
ORLD
OR 465.13  ; RK_07 U8_Z 铝壳上料移载Y轴JOG高速[M]
ANDLD
ANDNOT 765.14  ; RK_07 U8_Z 铝壳上料移载Y轴JOG低速[SW]
ANDNOT 365.14  ; RK_07 U8_Z 铝壳上料移载Y轴JOG低速[Pls]
OUT 465.13  ; RK_07 U8_Z 铝壳上料移载Y轴JOG高速[M]
LD TR0
AND 465.13  ; RK_07 U8_Z 铝壳上料移载Y轴JOG高速[M]
OUT 965.13  ; RK_07 U8_Z 铝壳上料移载Y轴JOG高速[lamp]
LD TR0
AND 765.14  ; RK_07 U8_Z 铝壳上料移载Y轴JOG低速[SW]
DIFU(013) 365.14  ; RK_07 U8_Z 铝壳上料移载Y轴JOG低速[Pls]
LD TR0
LD 365.14  ; RK_07 U8_Z 铝壳上料移载Y轴JOG低速[Pls]
OR 465.14  ; RK_07 U8_Z 铝壳上料移载Y轴JOG低速[M]
ANDLD
ANDNOT 765.13  ; RK_07 U8_Z 铝壳上料移载Y轴JOG高速[SW]
ANDNOT 365.13  ; RK_07 U8_Z 铝壳上料移载Y轴JOG高速[Pls]
OUT 465.14  ; RK_07 U8_Z 铝壳上料移载Y轴JOG低速[M]
LD TR0
AND 465.14  ; RK_07 U8_Z 铝壳上料移载Y轴JOG低速[M]
OUT 965.14  ; RK_07 U8_Z 铝壳上料移载Y轴JOG低速[lamp]

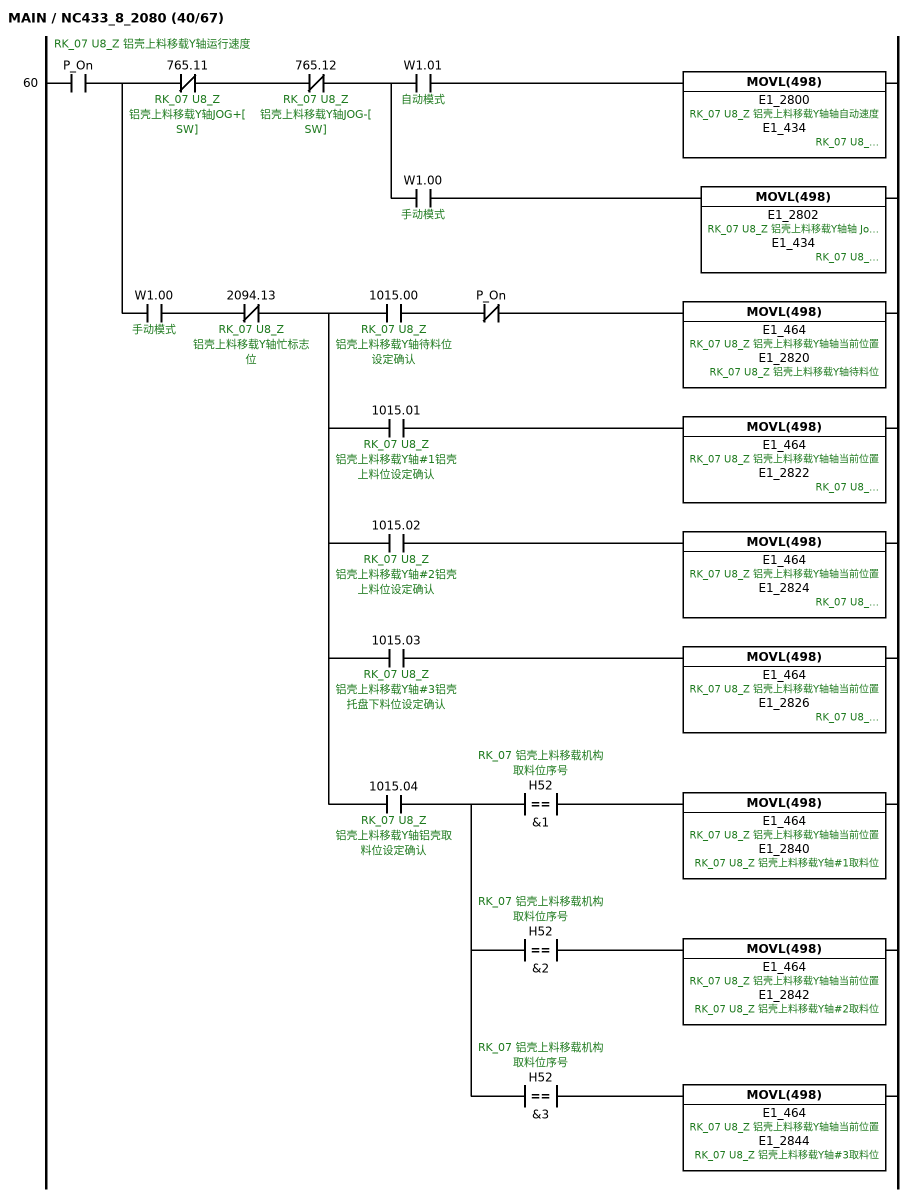
; rung 60: RK_07 U8_Z 铝壳上料移载Y轴运行速度
LD P_On
OUT TR0
ANDNOT 765.11  ; RK_07 U8_Z 铝壳上料移载Y轴JOG+[SW]
ANDNOT 765.12  ; RK_07 U8_Z 铝壳上料移载Y轴JOG-[SW]
OUT TR1
AND W1.01  ; 自动模式
MOVL(498) E1_2800 E1_434  ; RK_07 U8_Z 铝壳上料移载Y轴轴自动速度, RK_07 U8_Z 铝壳上料移载Y轴轴直接操作速度
LD TR1
AND W1.00  ; 手动模式
MOVL(498) E1_2802 E1_434  ; RK_07 U8_Z 铝壳上料移载Y轴轴 Jog 高速, RK_07 U8_Z 铝壳上料移载Y轴轴直接操作速度
LD TR0
AND W1.00  ; 手动模式
ANDNOT 2094.13  ; RK_07 U8_Z 铝壳上料移载Y轴忙标志位
OUT TR0
AND 1015.00  ; RK_07 U8_Z 铝壳上料移载Y轴待料位设定确认
ANDNOT P_On
MOVL(498) E1_464 E1_2820  ; RK_07 U8_Z 铝壳上料移载Y轴轴当前位置, RK_07 U8_Z 铝壳上料移载Y轴待料位
LD TR0
AND 1015.01  ; RK_07 U8_Z 铝壳上料移载Y轴#1铝壳上料位设定确认
MOVL(498) E1_464 E1_2822  ; RK_07 U8_Z 铝壳上料移载Y轴轴当前位置, RK_07 U8_Z 铝壳上料移载Y轴#1铝壳上料位
LD TR0
AND 1015.02  ; RK_07 U8_Z 铝壳上料移载Y轴#2铝壳上料位设定确认
MOVL(498) E1_464 E1_2824  ; RK_07 U8_Z 铝壳上料移载Y轴轴当前位置, RK_07 U8_Z 铝壳上料移载Y轴#2铝壳上料位
LD TR0
AND 1015.03  ; RK_07 U8_Z 铝壳上料移载Y轴#3铝壳托盘下料位设定确认
MOVL(498) E1_464 E1_2826  ; RK_07 U8_Z 铝壳上料移载Y轴轴当前位置, RK_07 U8_Z 铝壳上料移载Y轴#3铝壳托盘下料位
LD TR0
AND 1015.04  ; RK_07 U8_Z 铝壳上料移载Y轴铝壳取料位设定确认
OUT TR0
AND=(300) H52 &1  ; RK_07 铝壳上料移载机构取料位序号
MOVL(498) E1_464 E1_2840  ; RK_07 U8_Z 铝壳上料移载Y轴轴当前位置, RK_07 U8_Z 铝壳上料移载Y轴#1取料位
LD TR0
AND=(300) H52 &2  ; RK_07 铝壳上料移载机构取料位序号
MOVL(498) E1_464 E1_2842  ; RK_07 U8_Z 铝壳上料移载Y轴轴当前位置, RK_07 U8_Z 铝壳上料移载Y轴#2取料位
LD TR0
AND=(300) H52 &3  ; RK_07 铝壳上料移载机构取料位序号
MOVL(498) E1_464 E1_2844  ; RK_07 U8_Z 铝壳上料移载Y轴轴当前位置, RK_07 U8_Z 铝壳上料移载Y轴#3取料位

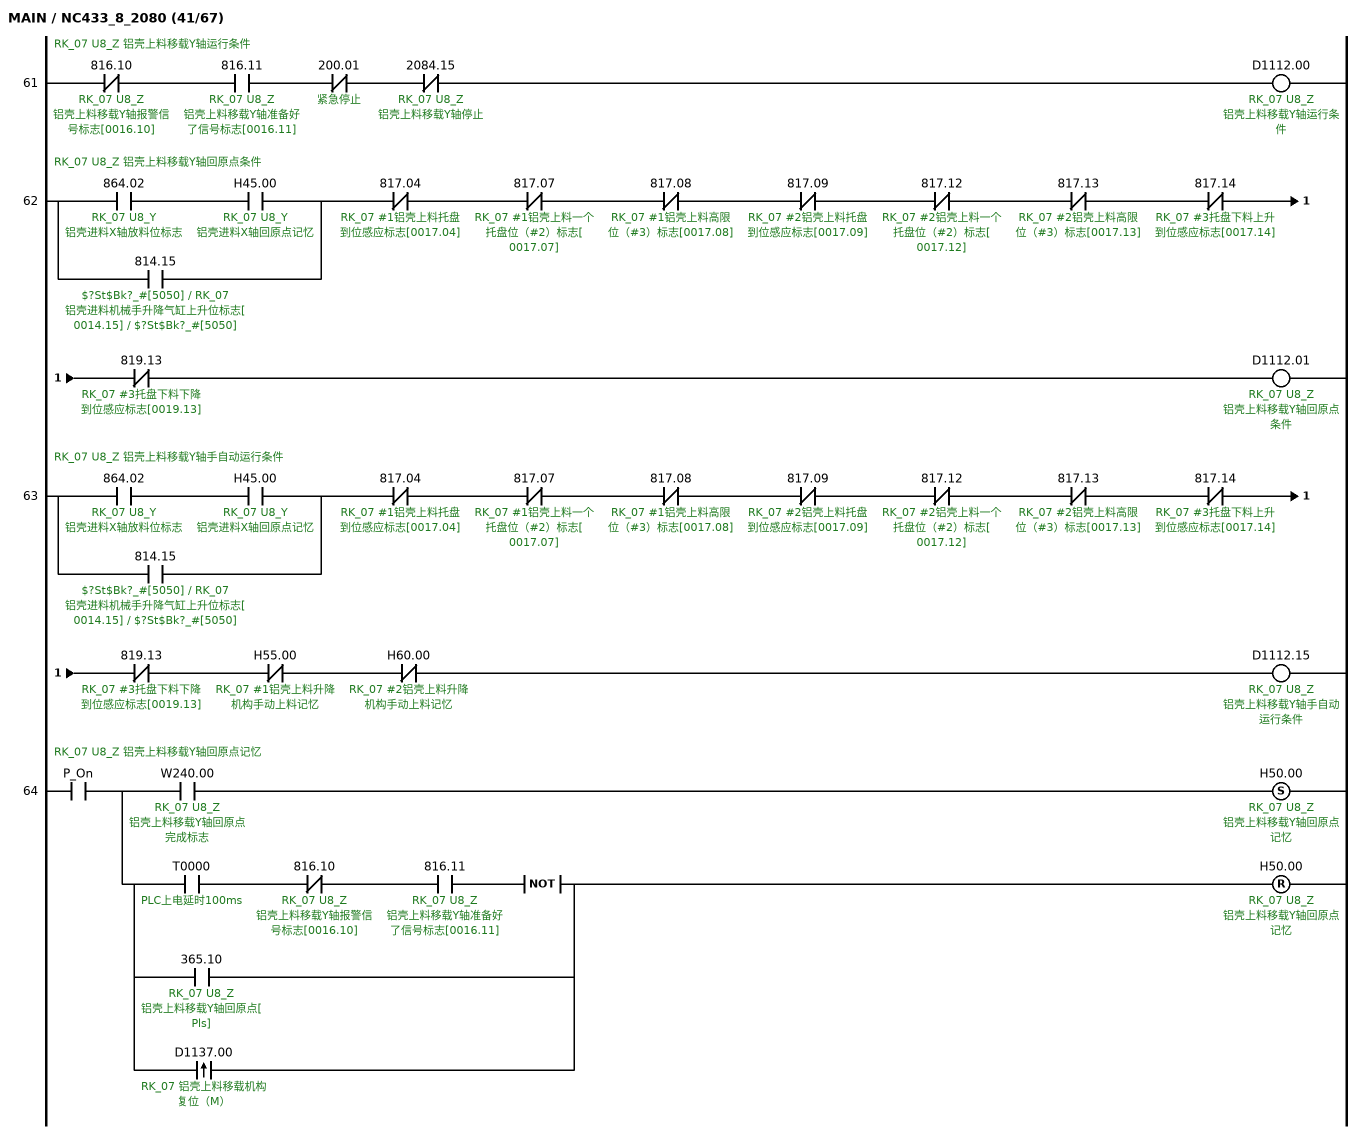
; rung 61: RK_07 U8_Z 铝壳上料移载Y轴运行条件
LDNOT 816.10  ; RK_07 U8_Z 铝壳上料移载Y轴报警信号标志[0016.10]
AND 816.11  ; RK_07 U8_Z 铝壳上料移载Y轴准备好了信号标志[0016.11]
ANDNOT 200.01  ; 紧急停止
ANDNOT 2084.15  ; RK_07 U8_Z 铝壳上料移载Y轴停止
OUT D1112.00  ; RK_07 U8_Z 铝壳上料移载Y轴运行条件
; rung 62: RK_07 U8_Z 铝壳上料移载Y轴回原点条件
LD 864.02  ; RK_07 U8_Y 铝壳进料X轴放料位标志
AND H45.00  ; RK_07 U8_Y 铝壳进料X轴回原点记忆
OR 814.15  ; $?St$Bk?_#[5050] / RK_07 铝壳进料机械手升降气缸上升位标志[0014.15] / $?St$Bk?_#[5050]
ANDNOT 817.04  ; RK_07 #1铝壳上料托盘到位感应标志[0017.04]
ANDNOT 817.07  ; RK_07 #1铝壳上料一个托盘位（#2）标志[0017.07]
ANDNOT 817.08  ; RK_07 #1铝壳上料高限位（#3）标志[0017.08]
ANDNOT 817.09  ; RK_07 #2铝壳上料托盘到位感应标志[0017.09]
ANDNOT 817.12  ; RK_07 #2铝壳上料一个托盘位（#2）标志[0017.12]
ANDNOT 817.13  ; RK_07 #2铝壳上料高限位（#3）标志[0017.13]
ANDNOT 817.14  ; RK_07 #3托盘下料上升到位感应标志[0017.14]
ANDNOT 819.13  ; RK_07 #3托盘下料下降到位感应标志[0019.13]
OUT D1112.01  ; RK_07 U8_Z 铝壳上料移载Y轴回原点条件
; rung 63: RK_07 U8_Z 铝壳上料移载Y轴手自动运行条件
LD 864.02  ; RK_07 U8_Y 铝壳进料X轴放料位标志
AND H45.00  ; RK_07 U8_Y 铝壳进料X轴回原点记忆
OR 814.15  ; $?St$Bk?_#[5050] / RK_07 铝壳进料机械手升降气缸上升位标志[0014.15] / $?St$Bk?_#[5050]
ANDNOT 817.04  ; RK_07 #1铝壳上料托盘到位感应标志[0017.04]
ANDNOT 817.07  ; RK_07 #1铝壳上料一个托盘位（#2）标志[0017.07]
ANDNOT 817.08  ; RK_07 #1铝壳上料高限位（#3）标志[0017.08]
ANDNOT 817.09  ; RK_07 #2铝壳上料托盘到位感应标志[0017.09]
ANDNOT 817.12  ; RK_07 #2铝壳上料一个托盘位（#2）标志[0017.12]
ANDNOT 817.13  ; RK_07 #2铝壳上料高限位（#3）标志[0017.13]
ANDNOT 817.14  ; RK_07 #3托盘下料上升到位感应标志[0017.14]
ANDNOT 819.13  ; RK_07 #3托盘下料下降到位感应标志[0019.13]
ANDNOT H55.00  ; RK_07 #1铝壳上料升降机构手动上料记忆
ANDNOT H60.00  ; RK_07 #2铝壳上料升降机构手动上料记忆
OUT D1112.15  ; RK_07 U8_Z 铝壳上料移载Y轴手自动运行条件
; rung 64: RK_07 U8_Z 铝壳上料移载Y轴回原点记忆
LD P_On
OUT TR0
AND W240.00  ; RK_07 U8_Z 铝壳上料移载Y轴回原点完成标志
SET H50.00  ; RK_07 U8_Z 铝壳上料移载Y轴回原点记忆
LD TR0
LD T0000  ; PLC上电延时100ms
ANDNOT 816.10  ; RK_07 U8_Z 铝壳上料移载Y轴报警信号标志[0016.10]
AND 816.11  ; RK_07 U8_Z 铝壳上料移载Y轴准备好了信号标志[0016.11]
NOT(520)
OR 365.10  ; RK_07 U8_Z 铝壳上料移载Y轴回原点[Pls]
@OR D1137.00  ; RK_07 铝壳上料移载机构复位（M）
ANDLD
RSET H50.00  ; RK_07 U8_Z 铝壳上料移载Y轴回原点记忆

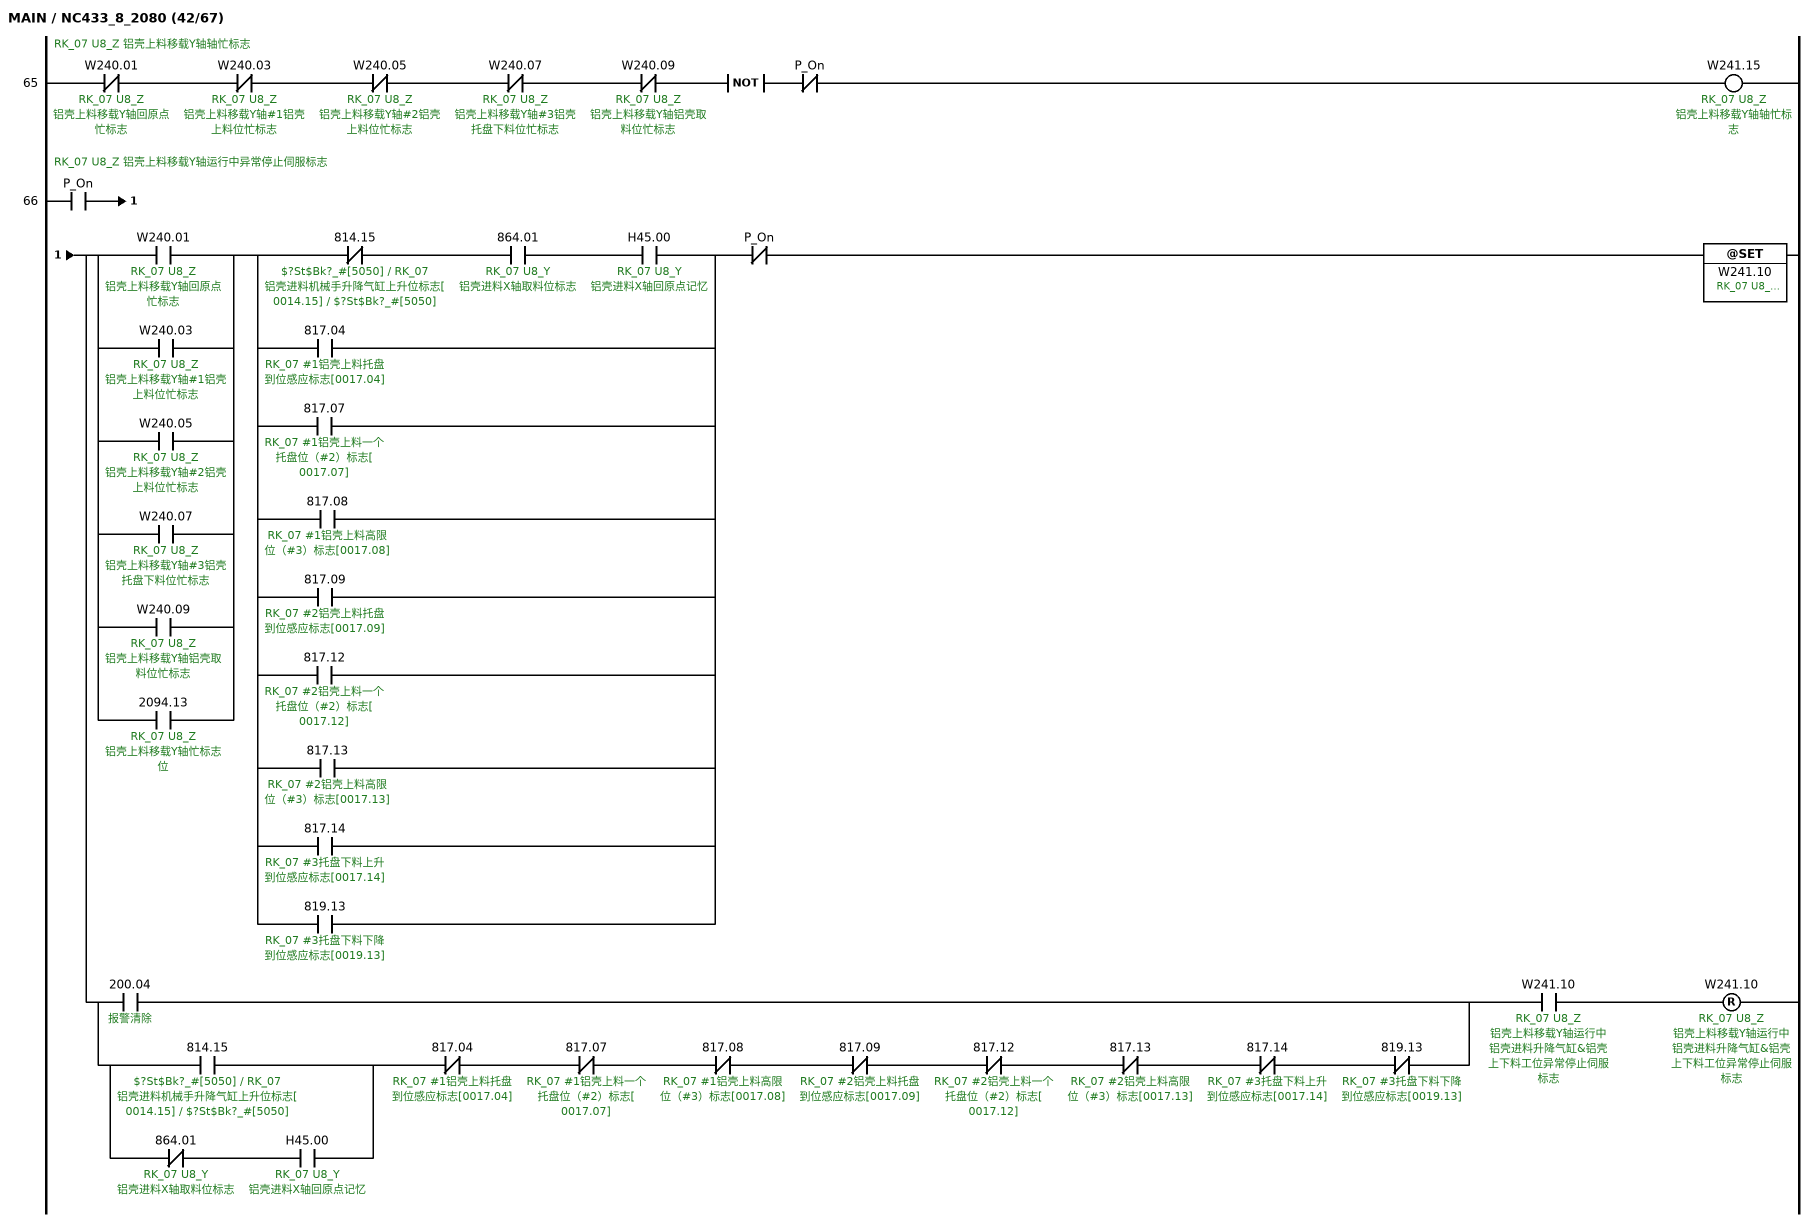
; rung 65: RK_07 U8_Z 铝壳上料移载Y轴轴忙标志
LDNOT W240.01  ; RK_07 U8_Z 铝壳上料移载Y轴回原点忙标志
ANDNOT W240.03  ; RK_07 U8_Z 铝壳上料移载Y轴#1铝壳上料位忙标志
ANDNOT W240.05  ; RK_07 U8_Z 铝壳上料移载Y轴#2铝壳上料位忙标志
ANDNOT W240.07  ; RK_07 U8_Z 铝壳上料移载Y轴#3铝壳托盘下料位忙标志
ANDNOT W240.09  ; RK_07 U8_Z 铝壳上料移载Y轴铝壳取料位忙标志
NOT(520)
ANDNOT P_On
OUT W241.15  ; RK_07 U8_Z 铝壳上料移载Y轴轴忙标志
; rung 66: RK_07 U8_Z 铝壳上料移载Y轴运行中异常停止伺服标志
LD P_On
OUT TR0
LD W240.01  ; RK_07 U8_Z 铝壳上料移载Y轴回原点忙标志
OR W240.03  ; RK_07 U8_Z 铝壳上料移载Y轴#1铝壳上料位忙标志
OR W240.05  ; RK_07 U8_Z 铝壳上料移载Y轴#2铝壳上料位忙标志
OR W240.07  ; RK_07 U8_Z 铝壳上料移载Y轴#3铝壳托盘下料位忙标志
OR W240.09  ; RK_07 U8_Z 铝壳上料移载Y轴铝壳取料位忙标志
OR 2094.13  ; RK_07 U8_Z 铝壳上料移载Y轴忙标志位
ANDLD
LDNOT 814.15  ; $?St$Bk?_#[5050] / RK_07 铝壳进料机械手升降气缸上升位标志[0014.15] / $?St$Bk?_#[5050]
AND 864.01  ; RK_07 U8_Y 铝壳进料X轴取料位标志
AND H45.00  ; RK_07 U8_Y 铝壳进料X轴回原点记忆
OR 817.04  ; RK_07 #1铝壳上料托盘到位感应标志[0017.04]
OR 817.07  ; RK_07 #1铝壳上料一个托盘位（#2）标志[0017.07]
OR 817.08  ; RK_07 #1铝壳上料高限位（#3）标志[0017.08]
OR 817.09  ; RK_07 #2铝壳上料托盘到位感应标志[0017.09]
OR 817.12  ; RK_07 #2铝壳上料一个托盘位（#2）标志[0017.12]
OR 817.13  ; RK_07 #2铝壳上料高限位（#3）标志[0017.13]
OR 817.14  ; RK_07 #3托盘下料上升到位感应标志[0017.14]
OR 819.13  ; RK_07 #3托盘下料下降到位感应标志[0019.13]
ANDLD
ANDNOT P_On
@SET W241.10  ; RK_07 U8_Z 铝壳上料移载Y轴运行中铝壳进料升降气缸&铝壳上下料工位异常停止伺服标志  // 增加相应报警信息
LD TR0
LD 200.04  ; 报警清除
LD 814.15  ; $?St$Bk?_#[5050] / RK_07 铝壳进料机械手升降气缸上升位标志[0014.15] / $?St$Bk?_#[5050]
LDNOT 864.01  ; RK_07 U8_Y 铝壳进料X轴取料位标志
AND H45.00  ; RK_07 U8_Y 铝壳进料X轴回原点记忆
ORLD
ANDNOT 817.04  ; RK_07 #1铝壳上料托盘到位感应标志[0017.04]
ANDNOT 817.07  ; RK_07 #1铝壳上料一个托盘位（#2）标志[0017.07]
ANDNOT 817.08  ; RK_07 #1铝壳上料高限位（#3）标志[0017.08]
ANDNOT 817.09  ; RK_07 #2铝壳上料托盘到位感应标志[0017.09]
ANDNOT 817.12  ; RK_07 #2铝壳上料一个托盘位（#2）标志[0017.12]
ANDNOT 817.13  ; RK_07 #2铝壳上料高限位（#3）标志[0017.13]
ANDNOT 817.14  ; RK_07 #3托盘下料上升到位感应标志[0017.14]
ANDNOT 819.13  ; RK_07 #3托盘下料下降到位感应标志[0019.13]
ORLD
ANDLD
AND W241.10  ; RK_07 U8_Z 铝壳上料移载Y轴运行中铝壳进料升降气缸&铝壳上下料工位异常停止伺服标志
RSET W241.10  ; RK_07 U8_Z 铝壳上料移载Y轴运行中铝壳进料升降气缸&铝壳上下料工位异常停止伺服标志

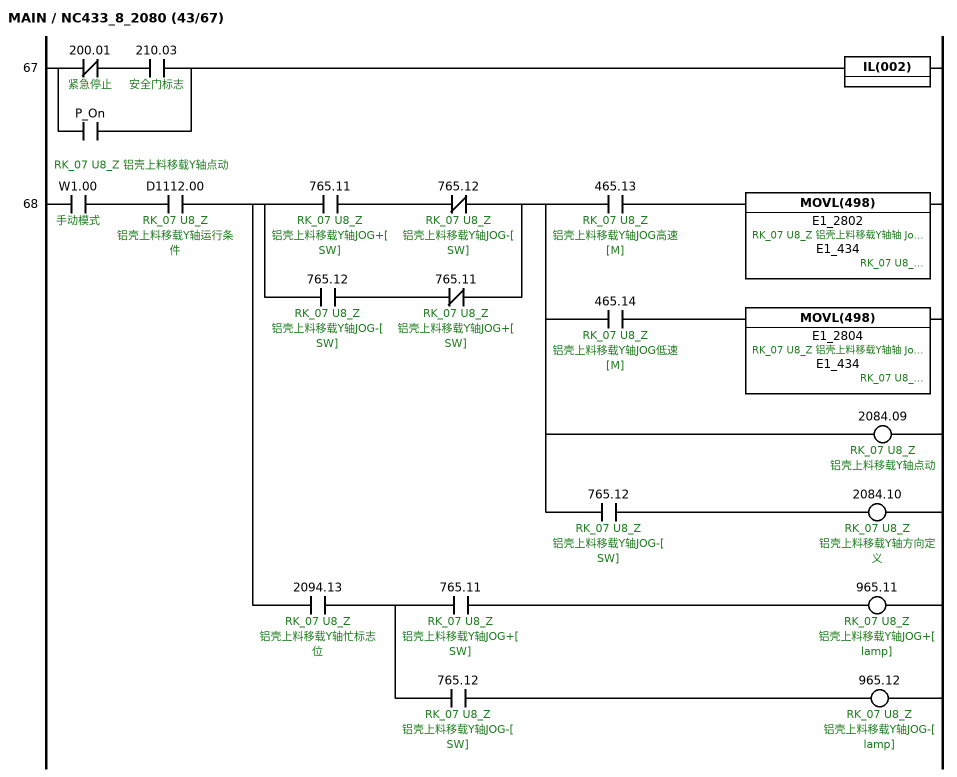
; rung 67
LDNOT 200.01  ; 紧急停止
AND 210.03  ; 安全门标志
OR P_On
IL(002)
; rung 68: RK_07 U8_Z 铝壳上料移载Y轴点动
LD W1.00  ; 手动模式
AND D1112.00  ; RK_07 U8_Z 铝壳上料移载Y轴运行条件
OUT TR0
LD 765.11  ; RK_07 U8_Z 铝壳上料移载Y轴JOG+[SW]
ANDNOT 765.12  ; RK_07 U8_Z 铝壳上料移载Y轴JOG-[SW]
LD 765.12  ; RK_07 U8_Z 铝壳上料移载Y轴JOG-[SW]
ANDNOT 765.11  ; RK_07 U8_Z 铝壳上料移载Y轴JOG+[SW]
ORLD
ANDLD
OUT TR1
AND 465.13  ; RK_07 U8_Z 铝壳上料移载Y轴JOG高速[M]
MOVL(498) E1_2802 E1_434  ; RK_07 U8_Z 铝壳上料移载Y轴轴 Jog 高速, RK_07 U8_Z 铝壳上料移载Y轴轴直接操作速度
LD TR1
AND 465.14  ; RK_07 U8_Z 铝壳上料移载Y轴JOG低速[M]
MOVL(498) E1_2804 E1_434  ; RK_07 U8_Z 铝壳上料移载Y轴轴 Jog 低速, RK_07 U8_Z 铝壳上料移载Y轴轴直接操作速度
LD TR1
OUT 2084.09  ; RK_07 U8_Z 铝壳上料移载Y轴点动
AND 765.12  ; RK_07 U8_Z 铝壳上料移载Y轴JOG-[SW]
OUT 2084.10  ; RK_07 U8_Z 铝壳上料移载Y轴方向定义
LD TR0
AND 2094.13  ; RK_07 U8_Z 铝壳上料移载Y轴忙标志位
OUT TR0
AND 765.11  ; RK_07 U8_Z 铝壳上料移载Y轴JOG+[SW]
OUT 965.11  ; RK_07 U8_Z 铝壳上料移载Y轴JOG+[lamp]
LD TR0
AND 765.12  ; RK_07 U8_Z 铝壳上料移载Y轴JOG-[SW]
OUT 965.12  ; RK_07 U8_Z 铝壳上料移载Y轴JOG-[lamp]

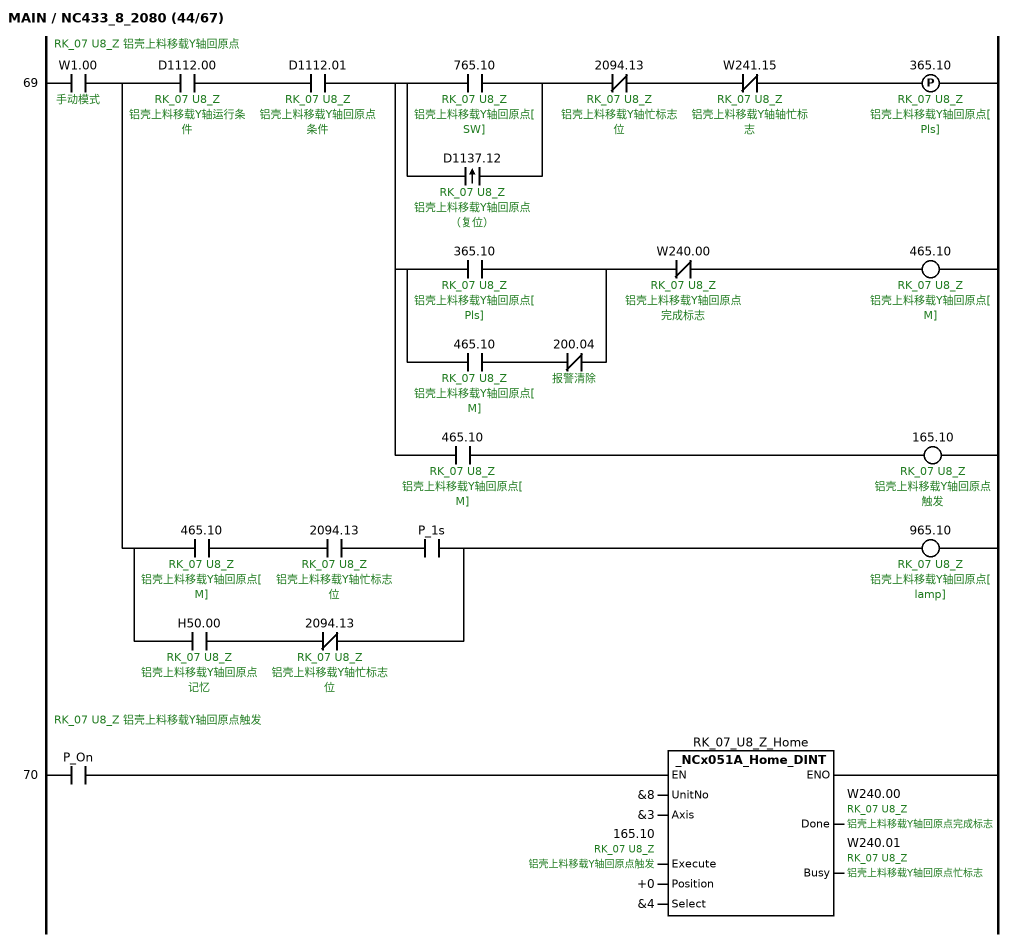
; rung 69: RK_07 U8_Z 铝壳上料移载Y轴回原点
LD W1.00  ; 手动模式
OUT TR0
AND D1112.00  ; RK_07 U8_Z 铝壳上料移载Y轴运行条件
AND D1112.01  ; RK_07 U8_Z 铝壳上料移载Y轴回原点条件
OUT TR1
LD 765.10  ; RK_07 U8_Z 铝壳上料移载Y轴回原点[SW]
@OR D1137.12  ; RK_07 U8_Z 铝壳上料移载Y轴回原点（复位）
ANDLD
ANDNOT 2094.13  ; RK_07 U8_Z 铝壳上料移载Y轴忙标志位
ANDNOT W241.15  ; RK_07 U8_Z 铝壳上料移载Y轴轴忙标志
DIFU(013) 365.10  ; RK_07 U8_Z 铝壳上料移载Y轴回原点[Pls]
LD TR1
LD 365.10  ; RK_07 U8_Z 铝壳上料移载Y轴回原点[Pls]
LD 465.10  ; RK_07 U8_Z 铝壳上料移载Y轴回原点[M]
ANDNOT 200.04  ; 报警清除
ORLD
ANDLD
ANDNOT W240.00  ; RK_07 U8_Z 铝壳上料移载Y轴回原点完成标志
OUT 465.10  ; RK_07 U8_Z 铝壳上料移载Y轴回原点[M]
LD TR1
AND 465.10  ; RK_07 U8_Z 铝壳上料移载Y轴回原点[M]
OUT 165.10  ; RK_07 U8_Z 铝壳上料移载Y轴回原点触发
LD TR0
LD 465.10  ; RK_07 U8_Z 铝壳上料移载Y轴回原点[M]
AND 2094.13  ; RK_07 U8_Z 铝壳上料移载Y轴忙标志位
AND P_1s
LD H50.00  ; RK_07 U8_Z 铝壳上料移载Y轴回原点记忆
ANDNOT 2094.13  ; RK_07 U8_Z 铝壳上料移载Y轴忙标志位
ORLD
ANDLD
OUT 965.10  ; RK_07 U8_Z 铝壳上料移载Y轴回原点[lamp]
; rung 70: RK_07 U8_Z 铝壳上料移载Y轴回原点触发
LD P_On
CALL RK_07_U8_Z_Home : _NCx051A_Home_DINT (UnitNo := &8, Axis := &3, Execute := 165.10, Position := +0, Select := &4, Done => W240.00, Busy => W240.01)  ; RK_07 U8_Z 铝壳上料移载Y轴回原点触发, RK_07 U8_Z 铝壳上料移载Y轴回原点完成标志, RK_07 U8_Z 铝壳上料移载Y轴回原点忙标志

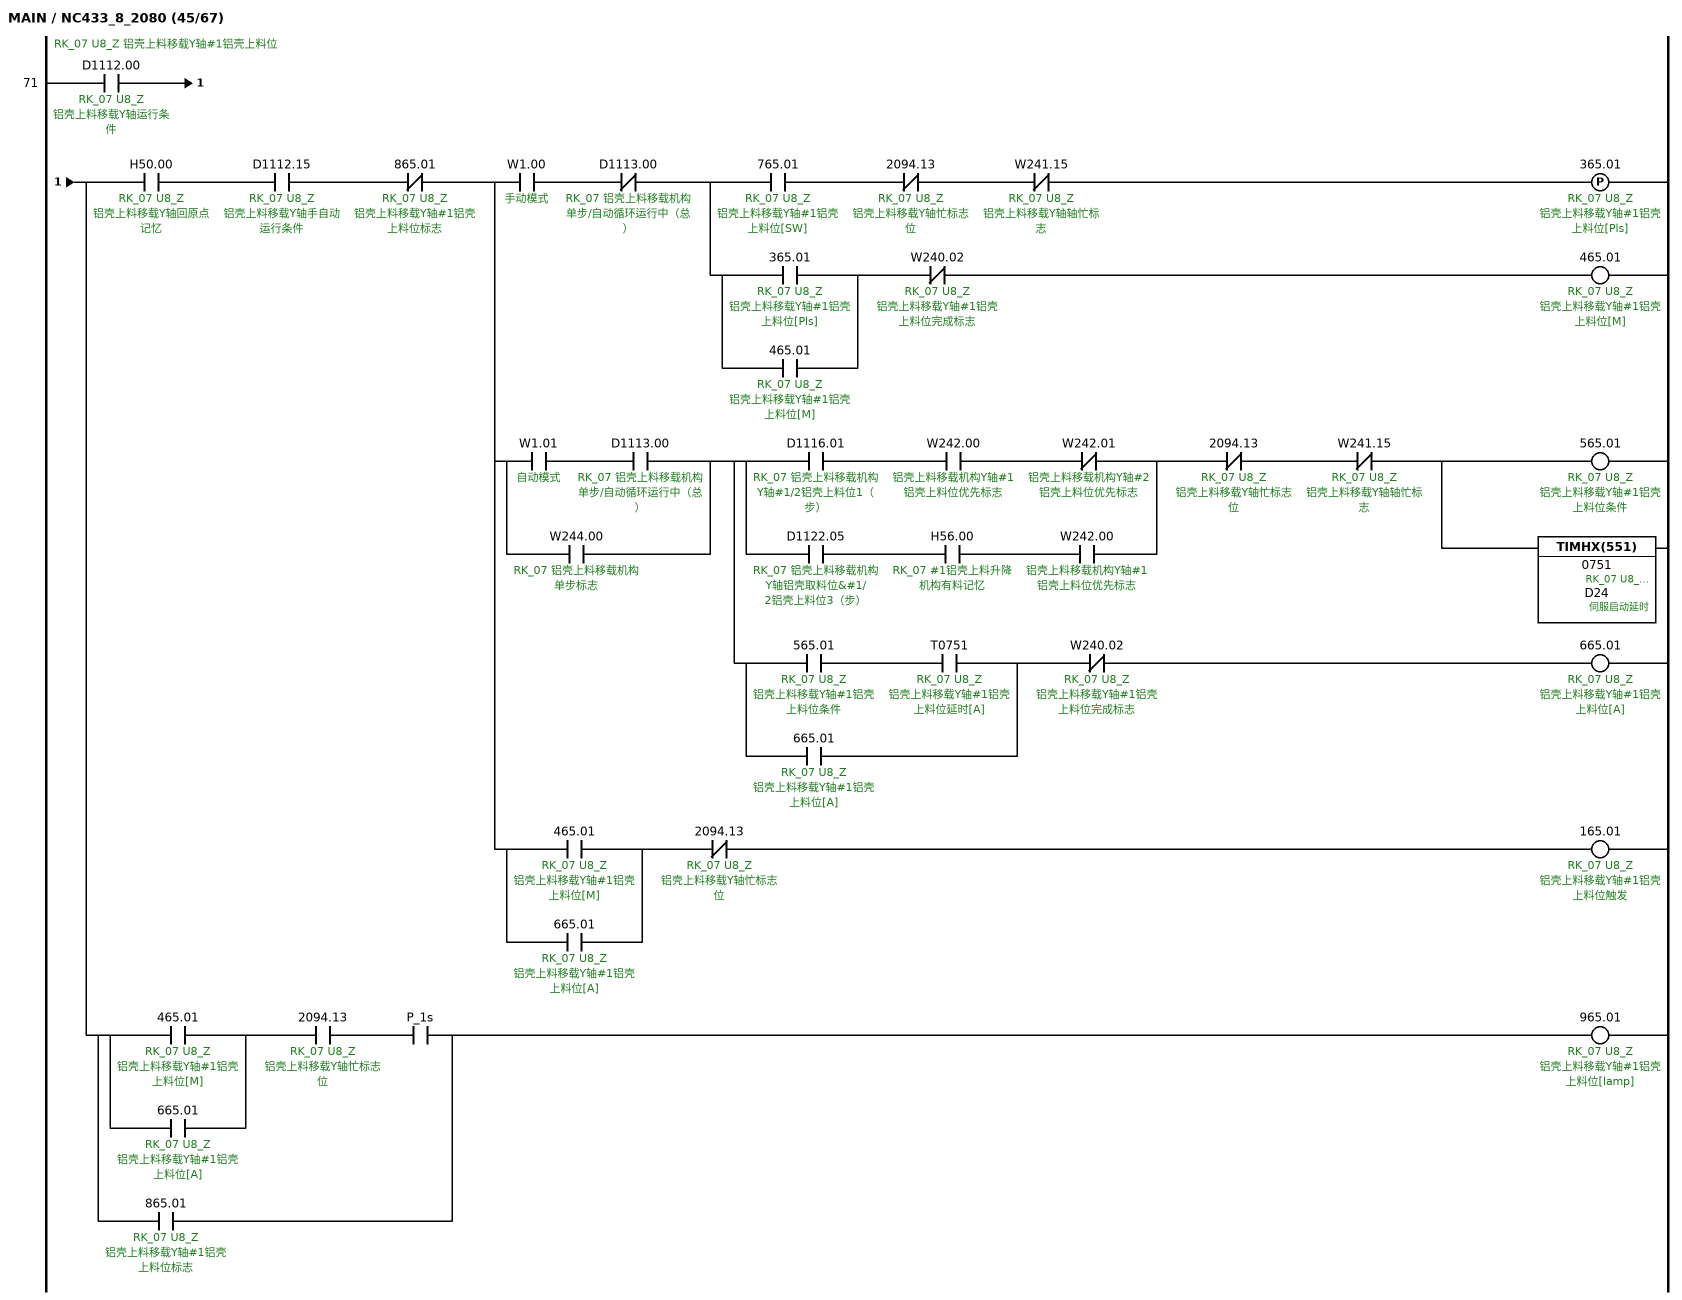
; rung 71: RK_07 U8_Z 铝壳上料移载Y轴#1铝壳上料位
LD D1112.00  ; RK_07 U8_Z 铝壳上料移载Y轴运行条件
OUT TR0
AND H50.00  ; RK_07 U8_Z 铝壳上料移载Y轴回原点记忆
AND D1112.15  ; RK_07 U8_Z 铝壳上料移载Y轴手自动运行条件
ANDNOT 865.01  ; RK_07 U8_Z 铝壳上料移载Y轴#1铝壳上料位标志
OUT TR1
AND W1.00  ; 手动模式
ANDNOT D1113.00  ; RK_07 铝壳上料移载机构单步/自动循环运行中（总）
OUT TR2
AND 765.01  ; RK_07 U8_Z 铝壳上料移载Y轴#1铝壳上料位[SW]
ANDNOT 2094.13  ; RK_07 U8_Z 铝壳上料移载Y轴忙标志位
ANDNOT W241.15  ; RK_07 U8_Z 铝壳上料移载Y轴轴忙标志
DIFU(013) 365.01  ; RK_07 U8_Z 铝壳上料移载Y轴#1铝壳上料位[Pls]
LD TR2
LD 365.01  ; RK_07 U8_Z 铝壳上料移载Y轴#1铝壳上料位[Pls]
OR 465.01  ; RK_07 U8_Z 铝壳上料移载Y轴#1铝壳上料位[M]
ANDLD
ANDNOT W240.02  ; RK_07 U8_Z 铝壳上料移载Y轴#1铝壳上料位完成标志
OUT 465.01  ; RK_07 U8_Z 铝壳上料移载Y轴#1铝壳上料位[M]
LD TR1
LD W1.01  ; 自动模式
AND D1113.00  ; RK_07 铝壳上料移载机构单步/自动循环运行中（总）
OR W244.00  ; RK_07 铝壳上料移载机构单步标志
ANDLD
OUT TR2
LD D1116.01  ; RK_07 铝壳上料移载机构Y轴#1/2铝壳上料位1（步）
AND W242.00  ; 铝壳上料移载机构Y轴#1铝壳上料位优先标志
ANDNOT W242.01  ; 铝壳上料移载机构Y轴#2铝壳上料位优先标志
LD D1122.05  ; RK_07 铝壳上料移载机构Y轴铝壳取料位&#1/2铝壳上料位3（步）
AND H56.00  ; RK_07 #1铝壳上料升降机构有料记忆
AND W242.00  ; 铝壳上料移载机构Y轴#1铝壳上料位优先标志
ORLD
ANDLD
ANDNOT 2094.13  ; RK_07 U8_Z 铝壳上料移载Y轴忙标志位
ANDNOT W241.15  ; RK_07 U8_Z 铝壳上料移载Y轴轴忙标志
OUT 565.01  ; RK_07 U8_Z 铝壳上料移载Y轴#1铝壳上料位条件
TIMHX(551) 0751 D24  ; 伺服启动延时, RK_07 U8_Z 铝壳上料移载Y轴#1铝壳上料位延时[A]
LD TR2
LD 565.01  ; RK_07 U8_Z 铝壳上料移载Y轴#1铝壳上料位条件
AND T0751  ; RK_07 U8_Z 铝壳上料移载Y轴#1铝壳上料位延时[A]
OR 665.01  ; RK_07 U8_Z 铝壳上料移载Y轴#1铝壳上料位[A]
ANDLD
ANDNOT W240.02  ; RK_07 U8_Z 铝壳上料移载Y轴#1铝壳上料位完成标志
OUT 665.01  ; RK_07 U8_Z 铝壳上料移载Y轴#1铝壳上料位[A]
LD TR1
LD 465.01  ; RK_07 U8_Z 铝壳上料移载Y轴#1铝壳上料位[M]
OR 665.01  ; RK_07 U8_Z 铝壳上料移载Y轴#1铝壳上料位[A]
ANDLD
ANDNOT 2094.13  ; RK_07 U8_Z 铝壳上料移载Y轴忙标志位
OUT 165.01  ; RK_07 U8_Z 铝壳上料移载Y轴#1铝壳上料位触发
LD TR0
LD 465.01  ; RK_07 U8_Z 铝壳上料移载Y轴#1铝壳上料位[M]
OR 665.01  ; RK_07 U8_Z 铝壳上料移载Y轴#1铝壳上料位[A]
AND 2094.13  ; RK_07 U8_Z 铝壳上料移载Y轴忙标志位
AND P_1s
OR 865.01  ; RK_07 U8_Z 铝壳上料移载Y轴#1铝壳上料位标志
ANDLD
OUT 965.01  ; RK_07 U8_Z 铝壳上料移载Y轴#1铝壳上料位[lamp]

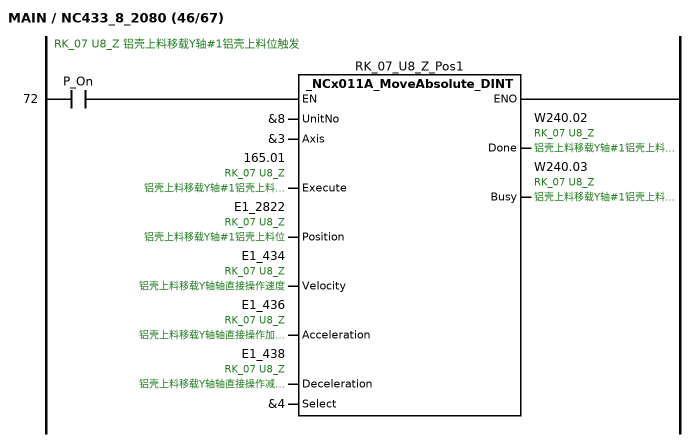
; rung 72: RK_07 U8_Z 铝壳上料移载Y轴#1铝壳上料位触发
LD P_On
CALL RK_07_U8_Z_Pos1 : _NCx011A_MoveAbsolute_DINT (UnitNo := &8, Axis := &3, Execute := 165.01, Position := E1_2822, Velocity := E1_434, Acceleration := E1_436, Deceleration := E1_438, Select := &4, Done => W240.02, Busy => W240.03)  ; RK_07 U8_Z 铝壳上料移载Y轴#1铝壳上料位触发, RK_07 U8_Z 铝壳上料移载Y轴#1铝壳上料位, RK_07 U8_Z 铝壳上料移载Y轴轴直接操作速度, RK_07 U8_Z 铝壳上料移载Y轴轴直接操作加速时间, RK_07 U8_Z 铝壳上料移载Y轴轴直接操作减速时间, RK_07 U8_Z 铝壳上料移载Y轴#1铝壳上料位完成标志, RK_07 U8_Z 铝壳上料移载Y轴#1铝壳上料位忙标志

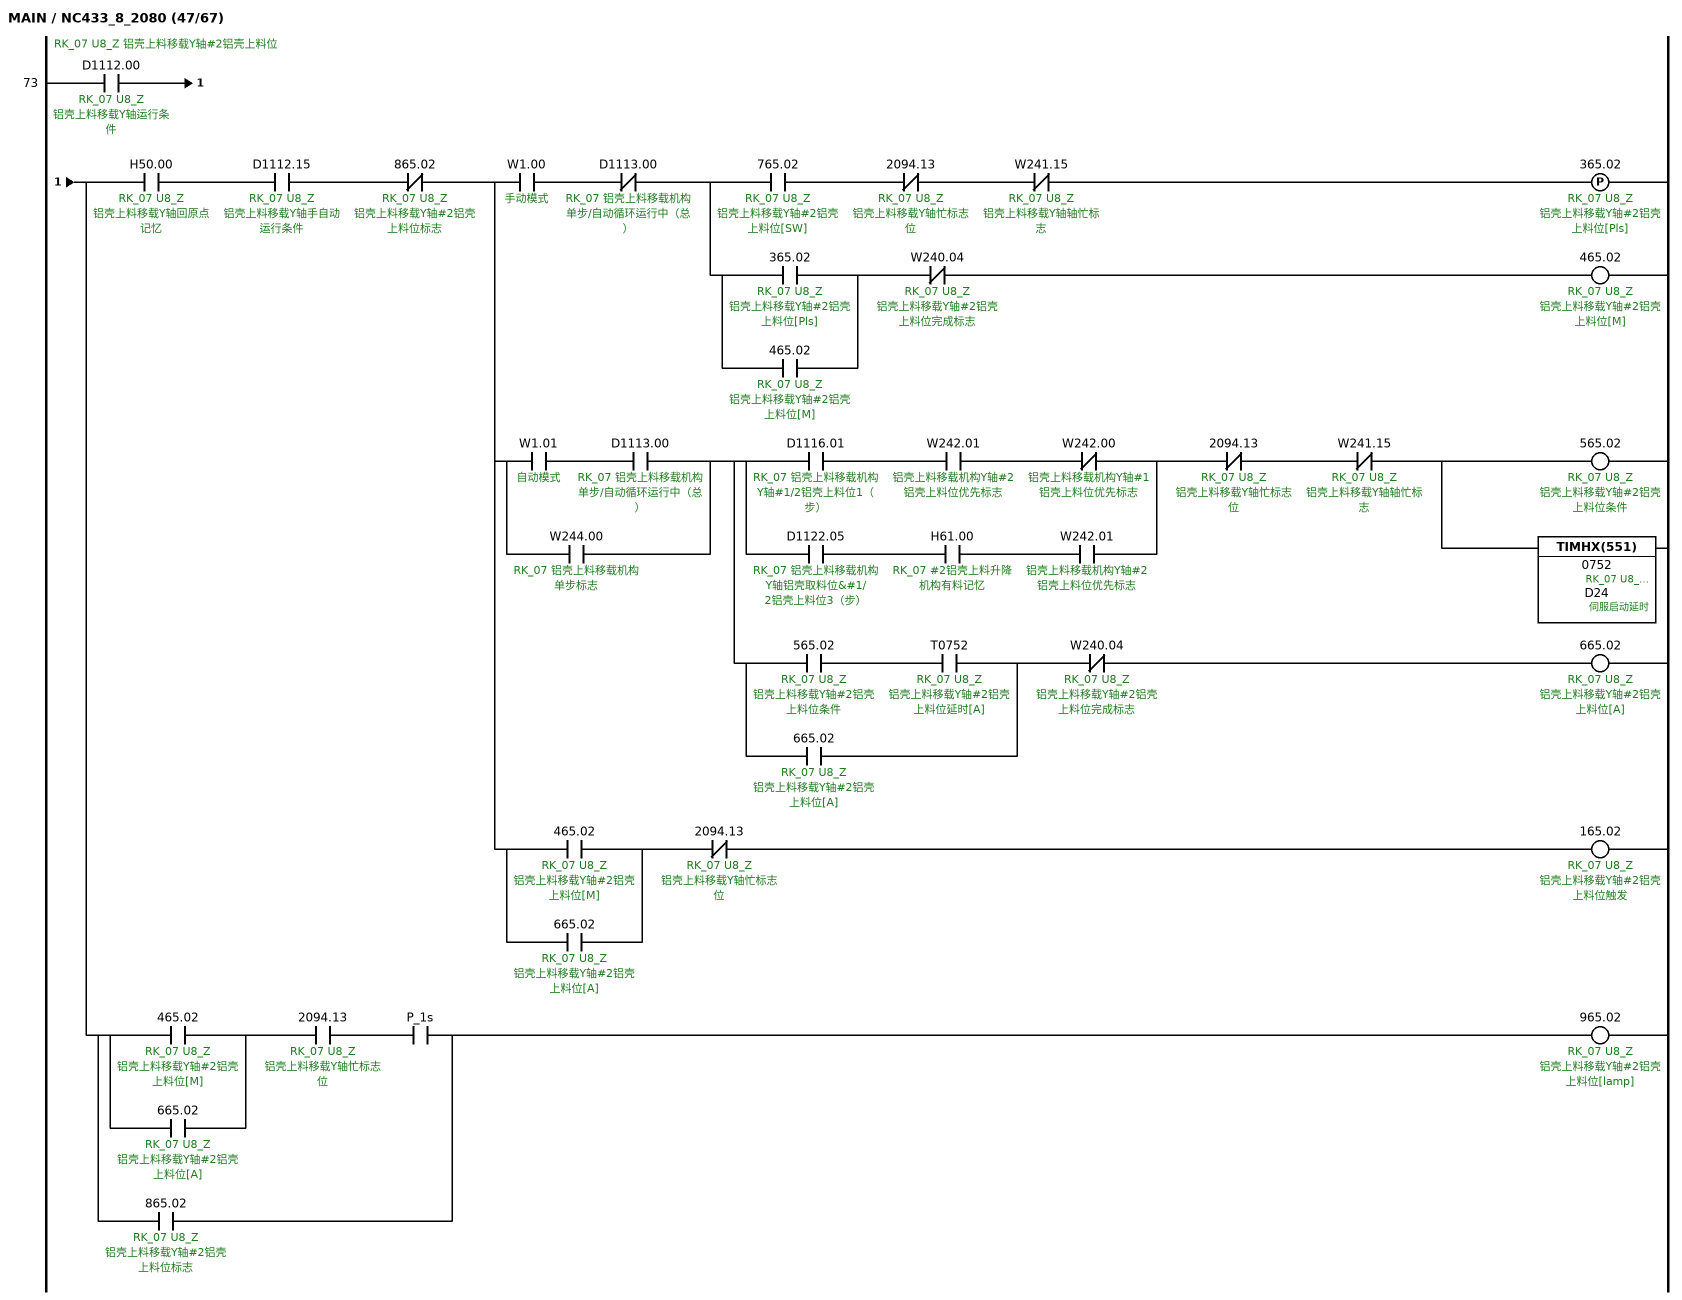
; rung 73: RK_07 U8_Z 铝壳上料移载Y轴#2铝壳上料位
LD D1112.00  ; RK_07 U8_Z 铝壳上料移载Y轴运行条件
OUT TR0
AND H50.00  ; RK_07 U8_Z 铝壳上料移载Y轴回原点记忆
AND D1112.15  ; RK_07 U8_Z 铝壳上料移载Y轴手自动运行条件
ANDNOT 865.02  ; RK_07 U8_Z 铝壳上料移载Y轴#2铝壳上料位标志
OUT TR1
AND W1.00  ; 手动模式
ANDNOT D1113.00  ; RK_07 铝壳上料移载机构单步/自动循环运行中（总）
OUT TR2
AND 765.02  ; RK_07 U8_Z 铝壳上料移载Y轴#2铝壳上料位[SW]
ANDNOT 2094.13  ; RK_07 U8_Z 铝壳上料移载Y轴忙标志位
ANDNOT W241.15  ; RK_07 U8_Z 铝壳上料移载Y轴轴忙标志
DIFU(013) 365.02  ; RK_07 U8_Z 铝壳上料移载Y轴#2铝壳上料位[Pls]
LD TR2
LD 365.02  ; RK_07 U8_Z 铝壳上料移载Y轴#2铝壳上料位[Pls]
OR 465.02  ; RK_07 U8_Z 铝壳上料移载Y轴#2铝壳上料位[M]
ANDLD
ANDNOT W240.04  ; RK_07 U8_Z 铝壳上料移载Y轴#2铝壳上料位完成标志
OUT 465.02  ; RK_07 U8_Z 铝壳上料移载Y轴#2铝壳上料位[M]
LD TR1
LD W1.01  ; 自动模式
AND D1113.00  ; RK_07 铝壳上料移载机构单步/自动循环运行中（总）
OR W244.00  ; RK_07 铝壳上料移载机构单步标志
ANDLD
OUT TR2
LD D1116.01  ; RK_07 铝壳上料移载机构Y轴#1/2铝壳上料位1（步）
AND W242.01  ; 铝壳上料移载机构Y轴#2铝壳上料位优先标志
ANDNOT W242.00  ; 铝壳上料移载机构Y轴#1铝壳上料位优先标志
LD D1122.05  ; RK_07 铝壳上料移载机构Y轴铝壳取料位&#1/2铝壳上料位3（步）
AND H61.00  ; RK_07 #2铝壳上料升降机构有料记忆
AND W242.01  ; 铝壳上料移载机构Y轴#2铝壳上料位优先标志
ORLD
ANDLD
ANDNOT 2094.13  ; RK_07 U8_Z 铝壳上料移载Y轴忙标志位
ANDNOT W241.15  ; RK_07 U8_Z 铝壳上料移载Y轴轴忙标志
OUT 565.02  ; RK_07 U8_Z 铝壳上料移载Y轴#2铝壳上料位条件
TIMHX(551) 0752 D24  ; 伺服启动延时, RK_07 U8_Z 铝壳上料移载Y轴#2铝壳上料位延时[A]
LD TR2
LD 565.02  ; RK_07 U8_Z 铝壳上料移载Y轴#2铝壳上料位条件
AND T0752  ; RK_07 U8_Z 铝壳上料移载Y轴#2铝壳上料位延时[A]
OR 665.02  ; RK_07 U8_Z 铝壳上料移载Y轴#2铝壳上料位[A]
ANDLD
ANDNOT W240.04  ; RK_07 U8_Z 铝壳上料移载Y轴#2铝壳上料位完成标志
OUT 665.02  ; RK_07 U8_Z 铝壳上料移载Y轴#2铝壳上料位[A]
LD TR1
LD 465.02  ; RK_07 U8_Z 铝壳上料移载Y轴#2铝壳上料位[M]
OR 665.02  ; RK_07 U8_Z 铝壳上料移载Y轴#2铝壳上料位[A]
ANDLD
ANDNOT 2094.13  ; RK_07 U8_Z 铝壳上料移载Y轴忙标志位
OUT 165.02  ; RK_07 U8_Z 铝壳上料移载Y轴#2铝壳上料位触发
LD TR0
LD 465.02  ; RK_07 U8_Z 铝壳上料移载Y轴#2铝壳上料位[M]
OR 665.02  ; RK_07 U8_Z 铝壳上料移载Y轴#2铝壳上料位[A]
AND 2094.13  ; RK_07 U8_Z 铝壳上料移载Y轴忙标志位
AND P_1s
OR 865.02  ; RK_07 U8_Z 铝壳上料移载Y轴#2铝壳上料位标志
ANDLD
OUT 965.02  ; RK_07 U8_Z 铝壳上料移载Y轴#2铝壳上料位[lamp]

